LIN {X 0,Y 482.021,Z 1133.799,A -85,B 0,C 180,E1 13794.402,E2 13794.402} C_VEL
LIN {X 0,Y 488.852,Z 1107.216,A -85,B 0,C 180,E1 13800.271,E2 13800.271} C_VEL
LIN {X 0,Y 497.315,Z 1077.498,A -85,B 0,C 180,E1 13805.263,E2 13805.263} C_VEL
LIN {X 0,Y 507.512,Z 1042.761,A -85,B 0,C 180,E1 13809.804,E2 13809.804} C_VEL
LIN {X 0,Y 518.482,Z 1004.016,A -85,B 0,C 180,E1 13813.68,E2 13813.68} C_VEL
LIN {X 0,Y 529.347,Z 962.337,A -85,B 0,C 180,E1 13816.876,E2 13816.876} C_VEL
LIN {X 0,Y 539.035,Z 917.758,A -85,B 0,C 180,E1 13819.437,E2 13819.437} C_VEL
LIN {X 0,Y 545.481,Z 880.736,A -85,B 0,C 180,E1 13821.049,E2 13821.049} C_VEL
LIN {X 0,Y 530.255,Z 846.769,A -85,B 0,C 180,E1 13825.083,E2 13825.083} C_VEL
LIN {X 0,Y 514.025,Z 818.402,A -85,B 0,C 180,E1 13829.146,E2 13829.146} C_VEL
LIN {X 0,Y 498.472,Z 795.623,A -85,B 0,C 180,E1 13833.243,E2 13833.243} C_VEL
LIN {X 0,Y 488.833,Z 782.735,A -85,B 0,C 180,E1 13836.078,E2 13836.078} C_VEL
LIN {X 0,Y 483.89,Z 776.161,A -85,B 0,C 180,E1 13837.704,E2 13837.704} C_VEL
LIN {X 0,Y 479.927,Z 770.269,A -85,B 0,C 180,E1 13839.148,E2 13839.148} C_VEL
LIN {X 0,Y 474.71,Z 764.689,A -85,B 0,C 180,E1 13841.152,E2 13841.152} C_VEL
LIN {X 0,Y 474.293,Z 762.06,A -85,B 0,C 180,E1 13841.534,E2 13841.534} C_VEL
LIN {X 0,Y 474.67,Z 762.06,A -85,B 0,C 180,E1 13847.136,E2 13847.136} C_VEL
LIN {X 0,Y 475.044,Z 762.06,A -85,B 0,C 180,E1 13853.146,E2 13853.146} C_VEL
LIN {X 0,Y 475.398,Z 762.06,A -85,B 0,C 180,E1 13858.189,E2 13858.189} C_VEL
LIN {X 0,Y 475.263,Z 762.06,A -85,B 0,C 180,E1 13863.656,E2 13863.656} C_VEL
LIN {X 0,Y 474.96,Z 762.06,A -85,B 0,C 180,E1 13869.496,E2 13869.496} C_VEL
LIN {X 0,Y 474.723,Z 762.06,A -85,B 0,C 180,E1 13874.762,E2 13874.762} C_VEL
LIN {X 0,Y 474.615,Z 762.484,A -85,B 0,C 180,E1 13878.205,E2 13878.205} C_VEL
LIN {X 0,Y 476.602,Z 767.385,A -85,B 0,C 180,E1 13879.126,E2 13879.126} C_VEL
LIN {X 0,Y 480.342,Z 770.702,A -85,B 0,C 180,E1 13880.495,E2 13880.495} C_VEL
LIN {X 0,Y 484.534,Z 776.398,A -85,B 0,C 180,E1 13881.986,E2 13881.986} C_VEL
LIN {X 0,Y 496.6,Z 792.603,A -85,B 0,C 180,E1 13885.705,E2 13885.705} C_VEL
LIN {X 0,Y 513.454,Z 816.532,A -85,B 0,C 180,E1 13890.028,E2 13890.028} C_VEL
LIN {X 0,Y 531.553,Z 846.468,A -85,B 0,C 180,E1 13894.197,E2 13894.197} C_VEL
LIN {X 0,Y 547.68,Z 879.498,A -85,B 0,C 180,E1 13897.952,E2 13897.952} C_VEL
LIN {X 0,Y 548.07,Z 883.694,A -85,B 0,C 180,E1 13898.206,E2 13898.206} C_VEL
LIN {X 0,Y 540.632,Z 928.209,A -85,B 0,C 180,E1 13899.828,E2 13899.828} C_VEL
LIN {X 0,Y 531.328,Z 973.235,A -85,B 0,C 180,E1 13902.174,E2 13902.174} C_VEL
LIN {X 0,Y 520.612,Z 1017.117,A -85,B 0,C 180,E1 13905.219,E2 13905.219} C_VEL
LIN {X 0,Y 510.113,Z 1056.037,A -85,B 0,C 180,E1 13908.767,E2 13908.767} C_VEL
LIN {X 0,Y 499.446,Z 1094.323,A -85,B 0,C 180,E1 13913.266,E2 13913.266} C_VEL
LIN {X 0,Y 490.54,Z 1126.605,A -85,B 0,C 180,E1 13918.183,E2 13918.183} C_VEL
LIN {X 0,Y 483.623,Z 1154.685,A -85,B 0,C 180,E1 13923.669,E2 13923.669} C_VEL
LIN {X 0,Y 479.218,Z 1176.457,A -85,B 0,C 180,E1 13929.307,E2 13929.307} C_VEL
LIN {X 0,Y 476.873,Z 1192.347,A -85,B 0,C 180,E1 13934.876,E2 13934.876} C_VEL
LIN {X 0,Y 475.804,Z 1202.186,A -85,B 0,C 180,E1 13939.929,E2 13939.929} C_VEL
LIN {X 0,Y 475.654,Z 1204.167,A -85,B 0,C 180,E1 13941.356,E2 13941.356} C_VEL
LIN {X 0,Y 473.042,Z 1206.128,A -85,B 0,C 180,E1 13942.887,E2 13942.887} C_VEL
LIN {X 0,Y 467.509,Z 1208.379,A -85,B 0,C 180,E1 13945.396,E2 13945.396} C_VEL
LIN {X 0,Y 467.504,Z 1208.319,A -85,B 0,C 180,E1 13945.463,E2 13945.463} C_VEL
LIN {X 0,Y 467.695,Z 1210,A -85,B 0,C 180,E1 13949.999,E2 13949.999} C_VEL
LIN {X 0,Y 467.612,Z 1207.633,A -85,B 0,C 180,E1 13955.562,E2 13955.562} C_VEL
LIN {X 0,Y 468.046,Z 1200.643,A -85,B 0,C 180,E1 13961.169,E2 13961.169} C_VEL
LIN {X 0,Y 469.482,Z 1188.604,A -85,B 0,C 180,E1 13966.838,E2 13966.838} C_VEL
LIN {X 0,Y 472.232,Z 1172.652,A -85,B 0,C 180,E1 13972.122,E2 13972.122} C_VEL
LIN {X 0,Y 477.422,Z 1149.519,A -85,B 0,C 180,E1 13977.829,E2 13977.829} C_VEL
LIN {X 0,Y 484.963,Z 1121.457,A -85,B 0,C 180,E1 13983.186,E2 13983.186} C_VEL
LIN {X 0,Y 494.517,Z 1087.969,A -85,B 0,C 180,E1 13988.108,E2 13988.108} C_VEL
LIN {X 0,Y 505.375,Z 1050.696,A -85,B 0,C 180,E1 13992.39,E2 13992.39} C_VEL
LIN {X 0,Y 516.934,Z 1008.902,A -85,B 0,C 180,E1 13996.039,E2 13996.039} C_VEL
LIN {X 0,Y 527.27,Z 967.405,A -85,B 0,C 180,E1 13998.822,E2 13998.822} C_VEL
LIN {X 0,Y 536.686,Z 921.282,A -85,B 0,C 180,E1 14001.121,E2 14001.121} C_VEL
LIN {X 0,Y 542.571,Z 883.848,A -85,B 0,C 180,E1 14002.522,E2 14002.522} C_VEL
LIN {X 0,Y 527.23,Z 851.526,A -85,B 0,C 180,E1 14006.303,E2 14006.303} C_VEL
LIN {X 0,Y 509.607,Z 821.901,A -85,B 0,C 180,E1 14010.564,E2 14010.564} C_VEL
LIN {X 0,Y 492.359,Z 797.074,A -85,B 0,C 180,E1 14015.213,E2 14015.213} C_VEL
LIN {X 0,Y 481.779,Z 783.224,A -85,B 0,C 180,E1 14018.607,E2 14018.607} C_VEL
LIN {X 0,Y 476.584,Z 776.309,A -85,B 0,C 180,E1 14020.545,E2 14020.545} C_VEL
LIN {X 0,Y 472.76,Z 771.079,A -85,B 0,C 180,E1 14022.135,E2 14022.135} C_VEL
LIN {X 0,Y 471.499,Z 769.36,A -85,B 0,C 180,E1 14022.696,E2 14022.696} C_VEL
LIN {X 0,Y 467.212,Z 764.911,A -85,B 0,C 180,E1 14024.695,E2 14024.695} C_VEL
LIN {X 0,Y 466.74,Z 762.06,A -85,B 0,C 180,E1 14025.152,E2 14025.152} C_VEL
LIN {X 0,Y 467.07,Z 762.06,A -85,B 0,C 180,E1 14030.681,E2 14030.681} C_VEL
LIN {X 0,Y 467.355,Z 762.06,A -85,B 0,C 180,E1 14036.282,E2 14036.282} C_VEL
LIN {X 0,Y 467.491,Z 762.06,A -85,B 0,C 180,E1 14041.841,E2 14041.841} C_VEL
LIN {X 0,Y 467.171,Z 762.06,A -85,B 0,C 180,E1 14047.422,E2 14047.422} C_VEL
LIN {X 0,Y 466.641,Z 762.06,A -85,B 0,C 180,E1 14053.72,E2 14053.72} C_VEL
LIN {X 0,Y 466.542,Z 762.875,A -85,B 0,C 180,E1 14055.305,E2 14055.305} C_VEL
LIN {X 0,Y 468.796,Z 767.622,A -85,B 0,C 180,E1 14056.55,E2 14056.55} C_VEL
LIN {X 0,Y 472.464,Z 770.774,A -85,B 0,C 180,E1 14058.157,E2 14058.157} C_VEL
LIN {X 0,Y 476.384,Z 776.273,A -85,B 0,C 180,E1 14059.803,E2 14059.803} C_VEL
LIN {X 0,Y 478.642,Z 779.134,A -85,B 0,C 180,E1 14060.669,E2 14060.669} C_VEL
LIN {X 0,Y 484.508,Z 786.882,A -85,B 0,C 180,E1 14062.75,E2 14062.75} C_VEL
LIN {X 0,Y 494.565,Z 800.367,A -85,B 0,C 180,E1 14065.895,E2 14065.895} C_VEL
LIN {X 0,Y 509.773,Z 823.065,A -85,B 0,C 180,E1 14070.123,E2 14070.123} C_VEL
LIN {X 0,Y 525.508,Z 851.418,A -85,B 0,C 180,E1 14074.276,E2 14074.276} C_VEL
LIN {X 0,Y 539.633,Z 883.823,A -85,B 0,C 180,E1 14078.242,E2 14078.242} C_VEL
LIN {X 0,Y 539.67,Z 888.681,A -85,B 0,C 180,E1 14078.535,E2 14078.535} C_VEL
LIN {X 0,Y 531.251,Z 930.768,A -85,B 0,C 180,E1 14080.477,E2 14080.477} C_VEL
LIN {X 0,Y 520.428,Z 975.76,A -85,B 0,C 180,E1 14083.297,E2 14083.297} C_VEL
LIN {X 0,Y 509.34,Z 1015.639,A -85,B 0,C 180,E1 14086.633,E2 14086.633} C_VEL
LIN {X 0,Y 497.817,Z 1054.175,A -85,B 0,C 180,E1 14090.841,E2 14090.841} C_VEL
LIN {X 0,Y 487.835,Z 1086.765,A -85,B 0,C 180,E1 14095.486,E2 14095.486} C_VEL
LIN {X 0,Y 479.242,Z 1116.664,A -85,B 0,C 180,E1 14101.002,E2 14101.002} C_VEL
LIN {X 0,Y 473.034,Z 1140.832,A -85,B 0,C 180,E1 14106.964,E2 14106.964} C_VEL
LIN {X 0,Y 469.704,Z 1158.095,A -85,B 0,C 180,E1 14112.688,E2 14112.688} C_VEL
LIN {X 0,Y 468.161,Z 1169.156,A -85,B 0,C 180,E1 14117.89,E2 14117.89} C_VEL
LIN {X 0,Y 467.701,Z 1175.956,A -85,B 0,C 180,E1 14122.575,E2 14122.575} C_VEL
LIN {X 0,Y 467.42,Z 1179.674,A -85,B 0,C 180,E1 14128.148,E2 14128.148} C_VEL
LIN {X 0,Y 467.598,Z 1179.656,A -85,B 0,C 180,E1 14131.853,E2 14131.853} C_VEL
LIN {X 0,Y 467.744,Z 1175.86,A -85,B 0,C 180,E1 14137.426,E2 14137.426} C_VEL
LIN {X 0,Y 468.381,Z 1167.229,A -85,B 0,C 180,E1 14143.053,E2 14143.053} C_VEL
LIN {X 0,Y 470.371,Z 1153.967,A -85,B 0,C 180,E1 14148.74,E2 14148.74} C_VEL
LIN {X 0,Y 474.261,Z 1135.424,A -85,B 0,C 180,E1 14154.471,E2 14154.471} C_VEL
LIN {X 0,Y 480.847,Z 1110.384,A -85,B 0,C 180,E1 14160.188,E2 14160.188} C_VEL
LIN {X 0,Y 489.563,Z 1081.41,A -85,B 0,C 180,E1 14165.278,E2 14165.278} C_VEL
LIN {X 0,Y 500.064,Z 1046.801,A -85,B 0,C 180,E1 14169.953,E2 14169.953} C_VEL
LIN {X 0,Y 511,Z 1010.288,A -85,B 0,C 180,E1 14173.776,E2 14173.776} C_VEL
LIN {X 0,Y 522.097,Z 969.271,A -85,B 0,C 180,E1 14177.06,E2 14177.06} C_VEL
LIN {X 0,Y 532.581,Z 924.406,A -85,B 0,C 180,E1 14179.779,E2 14179.779} C_VEL
LIN {X 0,Y 539.912,Z 884.236,A -85,B 0,C 180,E1 14181.599,E2 14181.599} C_VEL
LIN {X 0,Y 525.577,Z 851.517,A -85,B 0,C 180,E1 14185.604,E2 14185.604} C_VEL
LIN {X 0,Y 509.447,Z 822.562,A -85,B 0,C 180,E1 14189.851,E2 14189.851} C_VEL
LIN {X 0,Y 492.461,Z 797.228,A -85,B 0,C 180,E1 14194.62,E2 14194.62} C_VEL
LIN {X 0,Y 481.516,Z 783.139,A -85,B 0,C 180,E1 14198.134,E2 14198.134} C_VEL
LIN {X 0,Y 476.61,Z 776.434,A -85,B 0,C 180,E1 14199.965,E2 14199.965} C_VEL
LIN {X 0,Y 472.601,Z 771.322,A -85,B 0,C 180,E1 14201.608,E2 14201.608} C_VEL
LIN {X 0,Y 471.105,Z 769.289,A -85,B 0,C 180,E1 14202.272,E2 14202.272} C_VEL
LIN {X 0,Y 466.951,Z 764.704,A -85,B 0,C 180,E1 14204.228,E2 14204.228} C_VEL
LIN {X 0,Y 466.521,Z 762.06,A -85,B 0,C 180,E1 14204.754,E2 14204.754} C_VEL
LIN {X 0,Y 467.085,Z 762.06,A -85,B 0,C 180,E1 14210.703,E2 14210.703} C_VEL
LIN {X 0,Y 467.468,Z 762.06,A -85,B 0,C 180,E1 14216.304,E2 14216.304} C_VEL
LIN {X 0,Y 467.528,Z 762.06,A -85,B 0,C 180,E1 14221.863,E2 14221.863} C_VEL
LIN {X 0,Y 467.151,Z 762.06,A -85,B 0,C 180,E1 14227.444,E2 14227.444} C_VEL
LIN {X 0,Y 466.808,Z 762.06,A -85,B 0,C 180,E1 14233.796,E2 14233.796} C_VEL
LIN {X 0,Y 466.809,Z 762.508,A -85,B 0,C 180,E1 14235.078,E2 14235.078} C_VEL
LIN {X 0,Y 468.581,Z 767.145,A -85,B 0,C 180,E1 14236.098,E2 14236.098} C_VEL
LIN {X 0,Y 472.763,Z 770.814,A -85,B 0,C 180,E1 14237.921,E2 14237.921} C_VEL
LIN {X 0,Y 476.444,Z 776.177,A -85,B 0,C 180,E1 14239.461,E2 14239.461} C_VEL
LIN {X 0,Y 478.596,Z 778.637,A -85,B 0,C 180,E1 14240.271,E2 14240.271} C_VEL
LIN {X 0,Y 484.917,Z 787.333,A -85,B 0,C 180,E1 14242.51,E2 14242.51} C_VEL
LIN {X 0,Y 494.366,Z 799.789,A -85,B 0,C 180,E1 14245.405,E2 14245.405} C_VEL
LIN {X 0,Y 510.644,Z 823.428,A -85,B 0,C 180,E1 14249.711,E2 14249.711} C_VEL
LIN {X 0,Y 527.987,Z 853.064,A -85,B 0,C 180,E1 14253.901,E2 14253.901} C_VEL
LIN {X 0,Y 542.933,Z 884.677,A -85,B 0,C 180,E1 14257.574,E2 14257.574} C_VEL
LIN {X 0,Y 535.142,Z 929.856,A -85,B 0,C 180,E1 14259.248,E2 14259.248} C_VEL
LIN {X 0,Y 525.063,Z 976.261,A -85,B 0,C 180,E1 14261.713,E2 14261.713} C_VEL
LIN {X 0,Y 514.211,Z 1019.181,A -85,B 0,C 180,E1 14264.76,E2 14264.76} C_VEL
LIN {X 0,Y 502.972,Z 1058.986,A -85,B 0,C 180,E1 14268.487,E2 14268.487} C_VEL
LIN {X 0,Y 492.202,Z 1096.115,A -85,B 0,C 180,E1 14272.969,E2 14272.969} C_VEL
LIN {X 0,Y 482.385,Z 1130.255,A -85,B 0,C 180,E1 14278.35,E2 14278.35} C_VEL
LIN {X 0,Y 475.817,Z 1155.975,A -85,B 0,C 180,E1 14283.6,E2 14283.6} C_VEL
LIN {X 0,Y 471.294,Z 1177.475,A -85,B 0,C 180,E1 14289.347,E2 14289.347} C_VEL
LIN {X 0,Y 468.888,Z 1193.647,A -85,B 0,C 180,E1 14295.215,E2 14295.215} C_VEL
LIN {X 0,Y 467.832,Z 1203.513,A -85,B 0,C 180,E1 14300.705,E2 14300.705} C_VEL
LIN {X 0,Y 467.504,Z 1208.319,A -85,B 0,C 180,E1 14305.463,E2 14305.463} C_VEL
LIN {X 0,Y 464.981,Z 1209.328,A -85,B 0,C 180,E1 14307.044,E2 14307.044} C_VEL
LIN {X 0,Y 459.785,Z 1209.902,A -85,B 0,C 180,E1 14309.422,E2 14309.422} C_VEL
LIN {X 0,Y 459.736,Z 1209.946,A -85,B 0,C 180,E1 14309.696,E2 14309.696} C_VEL
LIN {X 0,Y 459.672,Z 1208.874,A -85,B 0,C 180,E1 14313.769,E2 14313.769} C_VEL
LIN {X 0,Y 459.913,Z 1204.668,A -85,B 0,C 180,E1 14318.502,E2 14318.502} C_VEL
LIN {X 0,Y 460.737,Z 1195.374,A -85,B 0,C 180,E1 14324.073,E2 14324.073} C_VEL
LIN {X 0,Y 463.106,Z 1180.326,A -85,B 0,C 180,E1 14330.035,E2 14330.035} C_VEL
LIN {X 0,Y 467.49,Z 1159.685,A -85,B 0,C 180,E1 14335.871,E2 14335.871} C_VEL
LIN {X 0,Y 474.645,Z 1132.681,A -85,B 0,C 180,E1 14341.688,E2 14341.688} C_VEL
LIN {X 0,Y 484.107,Z 1100.414,A -85,B 0,C 180,E1 14346.965,E2 14346.965} C_VEL
LIN {X 0,Y 494.946,Z 1064.966,A -85,B 0,C 180,E1 14351.478,E2 14351.478} C_VEL
LIN {X 0,Y 507.001,Z 1023.879,A -85,B 0,C 180,E1 14355.476,E2 14355.476} C_VEL
LIN {X 0,Y 517.974,Z 982.943,A -85,B 0,C 180,E1 14358.536,E2 14358.536} C_VEL
LIN {X 0,Y 529.125,Z 934.201,A -85,B 0,C 180,E1 14361.211,E2 14361.211} C_VEL
LIN {X 0,Y 537.157,Z 887.442,A -85,B 0,C 180,E1 14363.086,E2 14363.086} C_VEL
LIN {X 0,Y 522.309,Z 855.549,A -85,B 0,C 180,E1 14366.916,E2 14366.916} C_VEL
LIN {X 0,Y 505.838,Z 827.369,A -85,B 0,C 180,E1 14371.135,E2 14371.135} C_VEL
LIN {X 0,Y 489.999,Z 804.007,A -85,B 0,C 180,E1 14375.571,E2 14375.571} C_VEL
LIN {X 0,Y 479.443,Z 790.095,A -85,B 0,C 180,E1 14379.043,E2 14379.043} C_VEL
LIN {X 0,Y 474.776,Z 783.74,A -85,B 0,C 180,E1 14380.83,E2 14380.83} C_VEL
LIN {X 0,Y 470.687,Z 777.697,A -85,B 0,C 180,E1 14382.595,E2 14382.595} C_VEL
LIN {X 0,Y 465.499,Z 772.049,A -85,B 0,C 180,E1 14385.056,E2 14385.056} C_VEL
LIN {X 0,Y 464.758,Z 769.685,A -85,B 0,C 180,E1 14385.538,E2 14385.538} C_VEL
LIN {X 0,Y 459.786,Z 765.515,A -85,B 0,C 180,E1 14388.437,E2 14388.437} C_VEL
LIN {X 0,Y 459.057,Z 762.06,A -85,B 0,C 180,E1 14389.32,E2 14389.32} C_VEL
LIN {X 0,Y 459.365,Z 762.06,A -85,B 0,C 180,E1 14394.326,E2 14394.326} C_VEL
LIN {X 0,Y 459.759,Z 762.06,A -85,B 0,C 180,E1 14399.989,E2 14399.989} C_VEL
LIN {X 0,Y 459.408,Z 762.06,A -85,B 0,C 180,E1 14405.651,E2 14405.651} C_VEL
LIN {X 0,Y 459.012,Z 762.388,A -85,B 0,C 180,E1 14411.259,E2 14411.259} C_VEL
LIN {X 0,Y 460.474,Z 766.901,A -85,B 0,C 180,E1 14412.484,E2 14412.484} C_VEL
LIN {X 0,Y 464.855,Z 770.601,A -85,B 0,C 180,E1 14414.98,E2 14414.98} C_VEL
LIN {X 0,Y 468.212,Z 775.992,A -85,B 0,C 180,E1 14416.752,E2 14416.752} C_VEL
LIN {X 0,Y 470.825,Z 778.622,A -85,B 0,C 180,E1 14417.92,E2 14417.92} C_VEL
LIN {X 0,Y 475.459,Z 784.284,A -85,B 0,C 180,E1 14419.843,E2 14419.843} C_VEL
LIN {X 0,Y 488.256,Z 802.049,A -85,B 0,C 180,E1 14424.377,E2 14424.377} C_VEL
LIN {X 0,Y 501.005,Z 820.808,A -85,B 0,C 180,E1 14428.215,E2 14428.215} C_VEL
LIN {X 0,Y 516.276,Z 847.033,A -85,B 0,C 180,E1 14432.492,E2 14432.492} C_VEL
LIN {X 0,Y 530.399,Z 877.971,A -85,B 0,C 180,E1 14436.566,E2 14436.566} C_VEL
LIN {X 0,Y 534.534,Z 889.963,A -85,B 0,C 180,E1 14437.908,E2 14437.908} C_VEL
LIN {X 0,Y 525.762,Z 932.379,A -85,B 0,C 180,E1 14439.886,E2 14439.886} C_VEL
LIN {X 0,Y 514.844,Z 976.225,A -85,B 0,C 180,E1 14442.655,E2 14442.655} C_VEL
LIN {X 0,Y 503.09,Z 1017.032,A -85,B 0,C 180,E1 14446.105,E2 14446.105} C_VEL
LIN {X 0,Y 491.121,Z 1055.632,A -85,B 0,C 180,E1 14450.383,E2 14450.383} C_VEL
LIN {X 0,Y 480.429,Z 1089.06,A -85,B 0,C 180,E1 14455.266,E2 14455.266} C_VEL
LIN {X 0,Y 472.214,Z 1116.276,A -85,B 0,C 180,E1 14460.379,E2 14460.379} C_VEL
LIN {X 0,Y 465.927,Z 1139.404,A -85,B 0,C 180,E1 14466.085,E2 14466.085} C_VEL
LIN {X 0,Y 462.151,Z 1157.539,A -85,B 0,C 180,E1 14472.077,E2 14472.077} C_VEL
LIN {X 0,Y 460.321,Z 1169.407,A -85,B 0,C 180,E1 14477.681,E2 14477.681} C_VEL
LIN {X 0,Y 459.807,Z 1176.007,A -85,B 0,C 180,E1 14482.447,E2 14482.447} C_VEL
LIN {X 0,Y 459.517,Z 1179.673,A -85,B 0,C 180,E1 14488.116,E2 14488.116} C_VEL
LIN {X 0,Y 459.691,Z 1179.656,A -85,B 0,C 180,E1 14491.885,E2 14491.885} C_VEL
LIN {X 0,Y 459.852,Z 1175.916,A -85,B 0,C 180,E1 14497.554,E2 14497.554} C_VEL
LIN {X 0,Y 460.564,Z 1167.494,A -85,B 0,C 180,E1 14503.279,E2 14503.279} C_VEL
LIN {X 0,Y 462.682,Z 1154.236,A -85,B 0,C 180,E1 14509.063,E2 14509.063} C_VEL
LIN {X 0,Y 466.844,Z 1135.695,A -85,B 0,C 180,E1 14514.886,E2 14514.886} C_VEL
LIN {X 0,Y 474.217,Z 1109.478,A -85,B 0,C 180,E1 14520.92,E2 14520.92} C_VEL
LIN {X 0,Y 483.373,Z 1079.927,A -85,B 0,C 180,E1 14526.108,E2 14526.108} C_VEL
LIN {X 0,Y 494.425,Z 1045.238,A -85,B 0,C 180,E1 14530.783,E2 14530.783} C_VEL
LIN {X 0,Y 505.798,Z 1008.274,A -85,B 0,C 180,E1 14534.619,E2 14534.619} C_VEL
LIN {X 0,Y 517.301,Z 967.146,A -85,B 0,C 180,E1 14537.88,E2 14537.88} C_VEL
LIN {X 0,Y 527.574,Z 924.051,A -85,B 0,C 180,E1 14540.474,E2 14540.474} C_VEL
LIN {X 0,Y 534.465,Z 887.885,A -85,B 0,C 180,E1 14542.141,E2 14542.141} C_VEL
LIN {X 0,Y 520.643,Z 855.794,A -85,B 0,C 180,E1 14546.175,E2 14546.175} C_VEL
LIN {X 0,Y 505.438,Z 827.967,A -85,B 0,C 180,E1 14550.414,E2 14550.414} C_VEL
LIN {X 0,Y 489.726,Z 803.978,A -85,B 0,C 180,E1 14555.035,E2 14555.035} C_VEL
LIN {X 0,Y 479.336,Z 790.149,A -85,B 0,C 180,E1 14558.515,E2 14558.515} C_VEL
LIN {X 0,Y 474.508,Z 783.671,A -85,B 0,C 180,E1 14560.358,E2 14560.358} C_VEL
LIN {X 0,Y 470.417,Z 777.61,A -85,B 0,C 180,E1 14562.125,E2 14562.125} C_VEL
LIN {X 0,Y 465.226,Z 771.897,A -85,B 0,C 180,E1 14564.59,E2 14564.59} C_VEL
LIN {X 0,Y 464.131,Z 769.564,A -85,B 0,C 180,E1 14565.239,E2 14565.239} C_VEL
LIN {X 0,Y 459.461,Z 765.025,A -85,B 0,C 180,E1 14568.03,E2 14568.03} C_VEL
LIN {X 0,Y 458.988,Z 762.06,A -85,B 0,C 180,E1 14568.62,E2 14568.62} C_VEL
LIN {X 0,Y 459.36,Z 762.06,A -85,B 0,C 180,E1 14574.348,E2 14574.348} C_VEL
LIN {X 0,Y 459.775,Z 762.06,A -85,B 0,C 180,E1 14580.011,E2 14580.011} C_VEL
LIN {X 0,Y 459.366,Z 762.06,A -85,B 0,C 180,E1 14585.674,E2 14585.674} C_VEL
LIN {X 0,Y 459.087,Z 762.498,A -85,B 0,C 180,E1 14591.04,E2 14591.04} C_VEL
LIN {X 0,Y 460.872,Z 767.231,A -85,B 0,C 180,E1 14592.435,E2 14592.435} C_VEL
LIN {X 0,Y 465.092,Z 770.623,A -85,B 0,C 180,E1 14594.768,E2 14594.768} C_VEL
LIN {X 0,Y 468.478,Z 776.017,A -85,B 0,C 180,E1 14596.523,E2 14596.523} C_VEL
LIN {X 0,Y 471.01,Z 778.412,A -85,B 0,C 180,E1 14597.633,E2 14597.633} C_VEL
LIN {X 0,Y 475.518,Z 784.176,A -85,B 0,C 180,E1 14599.5,E2 14599.5} C_VEL
LIN {X 0,Y 487.699,Z 800.88,A -85,B 0,C 180,E1 14603.761,E2 14603.761} C_VEL
LIN {X 0,Y 502.204,Z 821.682,A -85,B 0,C 180,E1 14607.938,E2 14607.938} C_VEL
LIN {X 0,Y 519.434,Z 850.037,A -85,B 0,C 180,E1 14612.35,E2 14612.35} C_VEL
LIN {X 0,Y 535.88,Z 884.202,A -85,B 0,C 180,E1 14616.579,E2 14616.579} C_VEL
LIN {X 0,Y 537.377,Z 889.447,A -85,B 0,C 180,E1 14617.054,E2 14617.054} C_VEL
LIN {X 0,Y 529.104,Z 934.2,A -85,B 0,C 180,E1 14618.792,E2 14618.792} C_VEL
LIN {X 0,Y 518.434,Z 981.141,A -85,B 0,C 180,E1 14621.361,E2 14621.361} C_VEL
LIN {X 0,Y 507.485,Z 1022.217,A -85,B 0,C 180,E1 14624.386,E2 14624.386} C_VEL
LIN {X 0,Y 495.904,Z 1061.61,A -85,B 0,C 180,E1 14628.161,E2 14628.161} C_VEL
LIN {X 0,Y 485.242,Z 1096.941,A -85,B 0,C 180,E1 14632.537,E2 14632.537} C_VEL
LIN {X 0,Y 475.31,Z 1129.981,A -85,B 0,C 180,E1 14637.823,E2 14637.823} C_VEL
LIN {X 0,Y 468.393,Z 1155.702,A -85,B 0,C 180,E1 14643.149,E2 14643.149} C_VEL
LIN {X 0,Y 463.612,Z 1177.205,A -85,B 0,C 180,E1 14648.989,E2 14648.989} C_VEL
LIN {X 0,Y 461.095,Z 1193.034,A -85,B 0,C 180,E1 14654.8,E2 14654.8} C_VEL
LIN {X 0,Y 459.94,Z 1203.419,A -85,B 0,C 180,E1 14660.544,E2 14660.544} C_VEL
LIN {X 0,Y 459.599,Z 1208.369,A -85,B 0,C 180,E1 14665.465,E2 14665.465} C_VEL
LIN {X 0,Y 459.736,Z 1209.946,A -85,B 0,C 180,E1 14669.696,E2 14669.696} C_VEL
LIN {X 0,Y 457.353,Z 1209.886,A -85,B 0,C 180,E1 14671.305,E2 14671.305} C_VEL
LIN {X 0,Y 451.771,Z 1208.578,A -85,B 0,C 180,E1 14673.995,E2 14673.995} C_VEL
LIN {X 0,Y 452.069,Z 1203.161,A -85,B 0,C 180,E1 14679.62,E2 14679.62} C_VEL
LIN {X 0,Y 453.258,Z 1192.772,A -85,B 0,C 180,E1 14685.468,E2 14685.468} C_VEL
LIN {X 0,Y 455.955,Z 1176.943,A -85,B 0,C 180,E1 14691.379,E2 14691.379} C_VEL
LIN {X 0,Y 460.984,Z 1155.429,A -85,B 0,C 180,E1 14697.316,E2 14697.316} C_VEL
LIN {X 0,Y 468.753,Z 1128.396,A -85,B 0,C 180,E1 14702.95,E2 14702.95} C_VEL
LIN {X 0,Y 479.163,Z 1095.224,A -85,B 0,C 180,E1 14708.279,E2 14708.279} C_VEL
LIN {X 0,Y 490.331,Z 1059.502,A -85,B 0,C 180,E1 14712.686,E2 14712.686} C_VEL
LIN {X 0,Y 502.865,Z 1018.462,A -85,B 0,C 180,E1 14716.586,E2 14716.586} C_VEL
LIN {X 0,Y 514.507,Z 975.337,A -85,B 0,C 180,E1 14719.666,E2 14719.666} C_VEL
LIN {X 0,Y 525.319,Z 928.259,A -85,B 0,C 180,E1 14722.167,E2 14722.167} C_VEL
LIN {X 0,Y 532.13,Z 891.783,A -85,B 0,C 180,E1 14723.562,E2 14723.562} C_VEL
LIN {X 0,Y 517.239,Z 859.358,A -85,B 0,C 180,E1 14727.587,E2 14727.587} C_VEL
LIN {X 0,Y 501.801,Z 832.39,A -85,B 0,C 180,E1 14731.756,E2 14731.756} C_VEL
LIN {X 0,Y 487.096,Z 810.37,A -85,B 0,C 180,E1 14736.082,E2 14736.082} C_VEL
LIN {X 0,Y 477.134,Z 796.971,A -85,B 0,C 180,E1 14739.482,E2 14739.482} C_VEL
LIN {X 0,Y 472.566,Z 790.771,A -85,B 0,C 180,E1 14741.282,E2 14741.282} C_VEL
LIN {X 0,Y 467.697,Z 784.149,A -85,B 0,C 180,E1 14743.448,E2 14743.448} C_VEL
LIN {X 0,Y 463.522,Z 778.425,A -85,B 0,C 180,E1 14745.597,E2 14745.597} C_VEL
LIN {X 0,Y 458.058,Z 772.051,A -85,B 0,C 180,E1 14748.995,E2 14748.995} C_VEL
LIN {X 0,Y 457.521,Z 769.809,A -85,B 0,C 180,E1 14749.524,E2 14749.524} C_VEL
LIN {X 0,Y 451.937,Z 764.768,A -85,B 0,C 180,E1 14755.194,E2 14755.194} C_VEL
LIN {X 0,Y 451.543,Z 762.06,A -85,B 0,C 180,E1 14756.632,E2 14756.632} C_VEL
LIN {X 0,Y 451.699,Z 762.06,A -85,B 0,C 180,E1 14761.906,E2 14761.906} C_VEL
LIN {X 0,Y 451.618,Z 762.689,A -85,B 0,C 180,E1 14764.306,E2 14764.306} C_VEL
LIN {X 0,Y 454.334,Z 768.286,A -85,B 0,C 180,E1 14768.331,E2 14768.331} C_VEL
LIN {X 0,Y 457.573,Z 770.624,A -85,B 0,C 180,E1 14770.994,E2 14770.994} C_VEL
LIN {X 0,Y 460.337,Z 775.756,A -85,B 0,C 180,E1 14773.03,E2 14773.03} C_VEL
LIN {X 0,Y 463.367,Z 778.452,A -85,B 0,C 180,E1 14774.747,E2 14774.747} C_VEL
LIN {X 0,Y 467.52,Z 784.178,A -85,B 0,C 180,E1 14776.898,E2 14776.898} C_VEL
LIN {X 0,Y 470.033,Z 787.867,A -85,B 0,C 180,E1 14778.072,E2 14778.072} C_VEL
LIN {X 0,Y 475.252,Z 794.403,A -85,B 0,C 180,E1 14780.216,E2 14780.216} C_VEL
LIN {X 0,Y 484.874,Z 807.458,A -85,B 0,C 180,E1 14783.704,E2 14783.704} C_VEL
LIN {X 0,Y 499.036,Z 829.015,A -85,B 0,C 180,E1 14788.176,E2 14788.176} C_VEL
LIN {X 0,Y 514.041,Z 856.405,A -85,B 0,C 180,E1 14792.616,E2 14792.616} C_VEL
LIN {X 0,Y 527.344,Z 887.392,A -85,B 0,C 180,E1 14796.697,E2 14796.697} C_VEL
LIN {X 0,Y 529.028,Z 893.334,A -85,B 0,C 180,E1 14797.354,E2 14797.354} C_VEL
LIN {X 0,Y 519.844,Z 936.207,A -85,B 0,C 180,E1 14799.411,E2 14799.411} C_VEL
LIN {X 0,Y 508.661,Z 979.359,A -85,B 0,C 180,E1 14802.199,E2 14802.199} C_VEL
LIN {X 0,Y 496.002,Z 1021.296,A -85,B 0,C 180,E1 14805.85,E2 14805.85} C_VEL
LIN {X 0,Y 484.409,Z 1057.183,A -85,B 0,C 180,E1 14809.935,E2 14809.935} C_VEL
LIN {X 0,Y 473.255,Z 1090.647,A -85,B 0,C 180,E1 14814.919,E2 14814.919} C_VEL
LIN {X 0,Y 464.451,Z 1118.672,A -85,B 0,C 180,E1 14820.358,E2 14820.358} C_VEL
LIN {X 0,Y 457.604,Z 1143.059,A -85,B 0,C 180,E1 14826.656,E2 14826.656} C_VEL
LIN {X 0,Y 454.028,Z 1159.737,A -85,B 0,C 180,E1 14832.571,E2 14832.571} C_VEL
LIN {X 0,Y 452.299,Z 1171.183,A -85,B 0,C 180,E1 14838.437,E2 14838.437} C_VEL
LIN {X 0,Y 451.735,Z 1177.933,A -85,B 0,C 180,E1 14844.241,E2 14844.241} C_VEL
LIN {X 0,Y 451.786,Z 1180.185,A -85,B 0,C 180,E1 14850.001,E2 14850.001} C_VEL
LIN {X 0,Y 451.79,Z 1177.85,A -85,B 0,C 180,E1 14855.76,E2 14855.76} C_VEL
LIN {X 0,Y 452.345,Z 1171.039,A -85,B 0,C 180,E1 14861.563,E2 14861.563} C_VEL
LIN {X 0,Y 454.107,Z 1159.528,A -85,B 0,C 180,E1 14867.428,E2 14867.428} C_VEL
LIN {X 0,Y 457.688,Z 1142.757,A -85,B 0,C 180,E1 14873.341,E2 14873.341} C_VEL
LIN {X 0,Y 464.471,Z 1118.251,A -85,B 0,C 180,E1 14879.659,E2 14879.659} C_VEL
LIN {X 0,Y 473.436,Z 1090.165,A -85,B 0,C 180,E1 14885.067,E2 14885.067} C_VEL
LIN {X 0,Y 484.835,Z 1056.067,A -85,B 0,C 180,E1 14890.115,E2 14890.115} C_VEL
LIN {X 0,Y 497.048,Z 1018.082,A -85,B 0,C 180,E1 14894.367,E2 14894.367} C_VEL
LIN {X 0,Y 508.943,Z 978.42,A -85,B 0,C 180,E1 14897.771,E2 14897.771} C_VEL
LIN {X 0,Y 520.354,Z 933.446,A -85,B 0,C 180,E1 14900.664,E2 14900.664} C_VEL
LIN {X 0,Y 529.063,Z 891.817,A -85,B 0,C 180,E1 14902.649,E2 14902.649} C_VEL
LIN {X 0,Y 515.431,Z 859.33,A -85,B 0,C 180,E1 14906.858,E2 14906.858} C_VEL
LIN {X 0,Y 500.559,Z 831.68,A -85,B 0,C 180,E1 14911.256,E2 14911.256} C_VEL
LIN {X 0,Y 486.455,Z 809.923,A -85,B 0,C 180,E1 14915.636,E2 14915.636} C_VEL
LIN {X 0,Y 477.024,Z 797.056,A -85,B 0,C 180,E1 14918.941,E2 14918.941} C_VEL
LIN {X 0,Y 472.438,Z 790.828,A -85,B 0,C 180,E1 14920.754,E2 14920.754} C_VEL
LIN {X 0,Y 467.422,Z 784.115,A -85,B 0,C 180,E1 14922.977,E2 14922.977} C_VEL
LIN {X 0,Y 463.348,Z 778.514,A -85,B 0,C 180,E1 14925.071,E2 14925.071} C_VEL
LIN {X 0,Y 457.809,Z 771.742,A -85,B 0,C 180,E1 14928.53,E2 14928.53} C_VEL
LIN {X 0,Y 457.239,Z 769.765,A -85,B 0,C 180,E1 14929.058,E2 14929.058} C_VEL
LIN {X 0,Y 451.946,Z 764.794,A -85,B 0,C 180,E1 14934.315,E2 14934.315} C_VEL
LIN {X 0,Y 451.546,Z 762.06,A -85,B 0,C 180,E1 14935.693,E2 14935.693} C_VEL
LIN {X 0,Y 451.725,Z 762.06,A -85,B 0,C 180,E1 14941.928,E2 14941.928} C_VEL
LIN {X 0,Y 451.532,Z 762.79,A -85,B 0,C 180,E1 14944.209,E2 14944.209} C_VEL
LIN {X 0,Y 454.746,Z 768.615,A -85,B 0,C 180,E1 14948.501,E2 14948.501} C_VEL
LIN {X 0,Y 457.722,Z 770.78,A -85,B 0,C 180,E1 14950.832,E2 14950.832} C_VEL
LIN {X 0,Y 460.675,Z 775.934,A -85,B 0,C 180,E1 14952.922,E2 14952.922} C_VEL
LIN {X 0,Y 463.569,Z 778.441,A -85,B 0,C 180,E1 14954.522,E2 14954.522} C_VEL
LIN {X 0,Y 467.791,Z 784.176,A -85,B 0,C 180,E1 14956.669,E2 14956.669} C_VEL
LIN {X 0,Y 470.332,Z 787.951,A -85,B 0,C 180,E1 14957.841,E2 14957.841} C_VEL
LIN {X 0,Y 475.32,Z 794.243,A -85,B 0,C 180,E1 14959.872,E2 14959.872} C_VEL
LIN {X 0,Y 485.543,Z 808.042,A -85,B 0,C 180,E1 14963.448,E2 14963.448} C_VEL
LIN {X 0,Y 500.855,Z 830.453,A -85,B 0,C 180,E1 14967.981,E2 14967.981} C_VEL
LIN {X 0,Y 517.186,Z 859.304,A -85,B 0,C 180,E1 14972.417,E2 14972.417} C_VEL
LIN {X 0,Y 532.101,Z 891.662,A -85,B 0,C 180,E1 14976.435,E2 14976.435} C_VEL
LIN {X 0,Y 522.978,Z 939.007,A -85,B 0,C 180,E1 14978.345,E2 14978.345} C_VEL
LIN {X 0,Y 512.26,Z 984.248,A -85,B 0,C 180,E1 14980.894,E2 14980.894} C_VEL
LIN {X 0,Y 500.414,Z 1026.622,A -85,B 0,C 180,E1 14984.124,E2 14984.124} C_VEL
LIN {X 0,Y 488.688,Z 1065.032,A -85,B 0,C 180,E1 14987.92,E2 14987.92} C_VEL
LIN {X 0,Y 477.159,Z 1101.161,A -85,B 0,C 180,E1 14992.585,E2 14992.585} C_VEL
LIN {X 0,Y 467.404,Z 1132.729,A -85,B 0,C 180,E1 14997.832,E2 14997.832} C_VEL
LIN {X 0,Y 459.99,Z 1159.407,A -85,B 0,C 180,E1 15003.672,E2 15003.672} C_VEL
LIN {X 0,Y 455.375,Z 1180.047,A -85,B 0,C 180,E1 15009.608,E2 15009.608} C_VEL
LIN {X 0,Y 452.873,Z 1195.566,A -85,B 0,C 180,E1 15015.905,E2 15015.905} C_VEL
LIN {X 0,Y 452.03,Z 1204.402,A -85,B 0,C 180,E1 15021.347,E2 15021.347} C_VEL
LIN {X 0,Y 451.775,Z 1208.683,A -85,B 0,C 180,E1 15026.163,E2 15026.163} C_VEL
LIN {X 0,Y 451.904,Z 1209.849,A -85,B 0,C 180,E1 15029.999,E2 15029.999} C_VEL
LIN {X 0,Y 451.771,Z 1208.578,A -85,B 0,C 180,E1 15033.995,E2 15033.995} C_VEL
LIN {X 0,Y 447.847,Z 1206.978,A -85,B 0,C 180,E1 15036.153,E2 15036.153} C_VEL
LIN {X 0,Y 444.052,Z 1204.723,A -85,B 0,C 180,E1 15038.337,E2 15038.337} C_VEL
LIN {X 0,Y 445.037,Z 1195.305,A -85,B 0,C 180,E1 15044.346,E2 15044.346} C_VEL
LIN {X 0,Y 447.419,Z 1181.158,A -85,B 0,C 180,E1 15050.253,E2 15050.253} C_VEL
LIN {X 0,Y 452.107,Z 1161.124,A -85,B 0,C 180,E1 15056.286,E2 15056.286} C_VEL
LIN {X 0,Y 459.978,Z 1133.837,A -85,B 0,C 180,E1 15062.437,E2 15062.437} C_VEL
LIN {X 0,Y 469.772,Z 1103.312,A -85,B 0,C 180,E1 15067.673,E2 15067.673} C_VEL
LIN {X 0,Y 482.013,Z 1066.392,A -85,B 0,C 180,E1 15072.559,E2 15072.559} C_VEL
LIN {X 0,Y 494.043,Z 1028.406,A -85,B 0,C 180,E1 15076.392,E2 15076.392} C_VEL
LIN {X 0,Y 506.496,Z 985.467,A -85,B 0,C 180,E1 15079.713,E2 15079.713} C_VEL
LIN {X 0,Y 517.77,Z 939.926,A -85,B 0,C 180,E1 15082.303,E2 15082.303} C_VEL
LIN {X 0,Y 526.466,Z 894.645,A -85,B 0,C 180,E1 15084.209,E2 15084.209} C_VEL
LIN {X 0,Y 511.773,Z 862.118,A -85,B 0,C 180,E1 15088.407,E2 15088.407} C_VEL
LIN {X 0,Y 496.475,Z 835.239,A -85,B 0,C 180,E1 15092.768,E2 15092.768} C_VEL
LIN {X 0,Y 481.383,Z 812.27,A -85,B 0,C 180,E1 15097.559,E2 15097.559} C_VEL
LIN {X 0,Y 470.794,Z 798.156,A -85,B 0,C 180,E1 15101.573,E2 15101.573} C_VEL
LIN {X 0,Y 465.769,Z 791.379,A -85,B 0,C 180,E1 15103.862,E2 15103.862} C_VEL
LIN {X 0,Y 461.764,Z 785.309,A -85,B 0,C 180,E1 15106.025,E2 15106.025} C_VEL
LIN {X 0,Y 456.764,Z 779.762,A -85,B 0,C 180,E1 15109.205,E2 15109.205} C_VEL
LIN {X 0,Y 455.588,Z 777.383,A -85,B 0,C 180,E1 15110.203,E2 15110.203} C_VEL
LIN {X 0,Y 450.687,Z 771.81,A -85,B 0,C 180,E1 15115.783,E2 15115.783} C_VEL
LIN {X 0,Y 450.245,Z 769.846,A -85,B 0,C 180,E1 15117.104,E2 15117.104} C_VEL
LIN {X 0,Y 450.547,Z 770.62,A -85,B 0,C 180,E1 15124.136,E2 15124.136} C_VEL
LIN {X 0,Y 453.651,Z 776.366,A -85,B 0,C 180,E1 15128.609,E2 15128.609} C_VEL
LIN {X 0,Y 456.27,Z 778.52,A -85,B 0,C 180,E1 15130.784,E2 15130.784} C_VEL
LIN {X 0,Y 459.769,Z 784.049,A -85,B 0,C 180,E1 15133.288,E2 15133.288} C_VEL
LIN {X 0,Y 461.953,Z 786.384,A -85,B 0,C 180,E1 15134.551,E2 15134.551} C_VEL
LIN {X 0,Y 467.961,Z 794.586,A -85,B 0,C 180,E1 15137.608,E2 15137.608} C_VEL
LIN {X 0,Y 473.463,Z 802.025,A -85,B 0,C 180,E1 15140.002,E2 15140.002} C_VEL
LIN {X 0,Y 483.182,Z 815.526,A -85,B 0,C 180,E1 15143.607,E2 15143.607} C_VEL
LIN {X 0,Y 496.748,Z 837.029,A -85,B 0,C 180,E1 15148.103,E2 15148.103} C_VEL
LIN {X 0,Y 510.886,Z 864.237,A -85,B 0,C 180,E1 15152.528,E2 15152.528} C_VEL
LIN {X 0,Y 523.643,Z 895.92,A -85,B 0,C 180,E1 15156.742,E2 15156.742} C_VEL
LIN {X 0,Y 513.522,Z 941.732,A -85,B 0,C 180,E1 15159.015,E2 15159.015} C_VEL
LIN {X 0,Y 502.051,Z 983.739,A -85,B 0,C 180,E1 15161.847,E2 15161.847} C_VEL
LIN {X 0,Y 489.29,Z 1024.394,A -85,B 0,C 180,E1 15165.471,E2 15165.471} C_VEL
LIN {X 0,Y 477.127,Z 1060.332,A -85,B 0,C 180,E1 15169.695,E2 15169.695} C_VEL
LIN {X 0,Y 465.619,Z 1093.774,A -85,B 0,C 180,E1 15174.828,E2 15174.828} C_VEL
LIN {X 0,Y 456.758,Z 1120.652,A -85,B 0,C 180,E1 15180.249,E2 15180.249} C_VEL
LIN {X 0,Y 450.113,Z 1143.324,A -85,B 0,C 180,E1 15186.244,E2 15186.244} C_VEL
LIN {X 0,Y 446.315,Z 1160.001,A -85,B 0,C 180,E1 15192.26,E2 15192.26} C_VEL
LIN {X 0,Y 444.466,Z 1171.445,A -85,B 0,C 180,E1 15198.231,E2 15198.231} C_VEL
LIN {X 0,Y 443.841,Z 1178.192,A -85,B 0,C 180,E1 15204.139,E2 15204.139} C_VEL
LIN {X 0,Y 443.888,Z 1180.444,A -85,B 0,C 180,E1 15210.001,E2 15210.001} C_VEL
LIN {X 0,Y 443.896,Z 1178.111,A -85,B 0,C 180,E1 15215.863,E2 15215.863} C_VEL
LIN {X 0,Y 444.359,Z 1172.819,A -85,B 0,C 180,E1 15220.781,E2 15220.781} C_VEL
LIN {X 0,Y 445.96,Z 1162.023,A -85,B 0,C 180,E1 15226.74,E2 15226.74} C_VEL
LIN {X 0,Y 449.788,Z 1144.935,A -85,B 0,C 180,E1 15233.175,E2 15233.175} C_VEL
LIN {X 0,Y 456.074,Z 1122.618,A -85,B 0,C 180,E1 15239.206,E2 15239.206} C_VEL
LIN {X 0,Y 465.323,Z 1094.728,A -85,B 0,C 180,E1 15244.916,E2 15244.916} C_VEL
LIN {X 0,Y 476.914,Z 1060.933,A -85,B 0,C 180,E1 15250.129,E2 15250.129} C_VEL
LIN {X 0,Y 488.971,Z 1025.547,A -85,B 0,C 180,E1 15254.312,E2 15254.312} C_VEL
LIN {X 0,Y 501.855,Z 984.253,A -85,B 0,C 180,E1 15258.019,E2 15258.019} C_VEL
LIN {X 0,Y 513.373,Z 942.04,A -85,B 0,C 180,E1 15260.88,E2 15260.88} C_VEL
LIN {X 0,Y 523.468,Z 895.231,A -85,B 0,C 180,E1 15263.234,E2 15263.234} C_VEL
LIN {X 0,Y 510.501,Z 863.529,A -85,B 0,C 180,E1 15267.477,E2 15267.477} C_VEL
LIN {X 0,Y 496.231,Z 836.265,A -85,B 0,C 180,E1 15271.939,E2 15271.939} C_VEL
LIN {X 0,Y 481.192,Z 812.439,A -85,B 0,C 180,E1 15276.967,E2 15276.967} C_VEL
LIN {X 0,Y 470.492,Z 798.037,A -85,B 0,C 180,E1 15281.097,E2 15281.097} C_VEL
LIN {X 0,Y 465.739,Z 791.543,A -85,B 0,C 180,E1 15283.278,E2 15283.278} C_VEL
LIN {X 0,Y 461.587,Z 785.405,A -85,B 0,C 180,E1 15285.497,E2 15285.497} C_VEL
LIN {X 0,Y 456.514,Z 779.476,A -85,B 0,C 180,E1 15288.739,E2 15288.739} C_VEL
LIN {X 0,Y 455.63,Z 777.417,A -85,B 0,C 180,E1 15289.502,E2 15289.502} C_VEL
LIN {X 0,Y 450.719,Z 772.03,A -85,B 0,C 180,E1 15294.782,E2 15294.782} C_VEL
LIN {X 0,Y 450.18,Z 769.822,A -85,B 0,C 180,E1 15296.162,E2 15296.162} C_VEL
LIN {X 0,Y 450.442,Z 770.521,A -85,B 0,C 180,E1 15303.978,E2 15303.978} C_VEL
LIN {X 0,Y 453.645,Z 776.387,A -85,B 0,C 180,E1 15308.39,E2 15308.39} C_VEL
LIN {X 0,Y 456.349,Z 778.445,A -85,B 0,C 180,E1 15310.564,E2 15310.564} C_VEL
LIN {X 0,Y 459.724,Z 783.883,A -85,B 0,C 180,E1 15312.949,E2 15312.949} C_VEL
LIN {X 0,Y 462.159,Z 786.277,A -85,B 0,C 180,E1 15314.325,E2 15314.325} C_VEL
LIN {X 0,Y 466.858,Z 792.113,A -85,B 0,C 180,E1 15316.703,E2 15316.703} C_VEL
LIN {X 0,Y 478.348,Z 808.124,A -85,B 0,C 180,E1 15321.409,E2 15321.409} C_VEL
LIN {X 0,Y 491.363,Z 827.011,A -85,B 0,C 180,E1 15325.692,E2 15325.692} C_VEL
LIN {X 0,Y 507.029,Z 853.129,A -85,B 0,C 180,E1 15330.271,E2 15330.271} C_VEL
LIN {X 0,Y 522.707,Z 885.469,A -85,B 0,C 180,E1 15334.698,E2 15334.698} C_VEL
LIN {X 0,Y 526.458,Z 896.483,A -85,B 0,C 180,E1 15335.914,E2 15335.914} C_VEL
LIN {X 0,Y 516.69,Z 944.806,A -85,B 0,C 180,E1 15337.938,E2 15337.938} C_VEL
LIN {X 0,Y 505.343,Z 989.525,A -85,B 0,C 180,E1 15340.574,E2 15340.574} C_VEL
LIN {X 0,Y 492.899,Z 1032.247,A -85,B 0,C 180,E1 15343.953,E2 15343.953} C_VEL
LIN {X 0,Y 480.883,Z 1069.691,A -85,B 0,C 180,E1 15347.838,E2 15347.838} C_VEL
LIN {X 0,Y 468.794,Z 1106.539,A -85,B 0,C 180,E1 15352.815,E2 15352.815} C_VEL
LIN {X 0,Y 458.946,Z 1137.031,A -85,B 0,C 180,E1 15358.209,E2 15358.209} C_VEL
LIN {X 0,Y 451.613,Z 1163.104,A -85,B 0,C 180,E1 15364.215,E2 15364.215} C_VEL
LIN {X 0,Y 447.161,Z 1182.521,A -85,B 0,C 180,E1 15370.248,E2 15370.248} C_VEL
LIN {X 0,Y 444.853,Z 1196.476,A -85,B 0,C 180,E1 15376.243,E2 15376.243} C_VEL
LIN {X 0,Y 444.053,Z 1205.363,A -85,B 0,C 180,E1 15382.176,E2 15382.176} C_VEL
LIN {X 0,Y 443.853,Z 1209.241,A -85,B 0,C 180,E1 15388.048,E2 15388.048} C_VEL
LIN {X 0,Y 444.048,Z 1209.248,A -85,B 0,C 180,E1 15391.949,E2 15391.949} C_VEL
LIN {X 0,Y 444.056,Z 1205.367,A -85,B 0,C 180,E1 15397.822,E2 15397.822} C_VEL
LIN {X 0,Y 444.052,Z 1204.723,A -85,B 0,C 180,E1 15398.337,E2 15398.337} C_VEL
LIN {X 0,Y 440.273,Z 1201.963,A -85,B 0,C 180,E1 15400.522,E2 15400.522} C_VEL
LIN {X 0,Y 436.686,Z 1198.48,A -85,B 0,C 180,E1 15402.736,E2 15402.736} C_VEL
LIN {X 0,Y 438.64,Z 1186.476,A -85,B 0,C 180,E1 15408.529,E2 15408.529} C_VEL
LIN {X 0,Y 442.934,Z 1167.536,A -85,B 0,C 180,E1 15414.894,E2 15414.894} C_VEL
LIN {X 0,Y 450.133,Z 1142.689,A -85,B 0,C 180,E1 15421.118,E2 15421.118} C_VEL
LIN {X 0,Y 460.111,Z 1112.311,A -85,B 0,C 180,E1 15426.824,E2 15426.824} C_VEL
LIN {X 0,Y 471.7,Z 1078.475,A -85,B 0,C 180,E1 15431.733,E2 15431.733} C_VEL
LIN {X 0,Y 485.208,Z 1038.055,A -85,B 0,C 180,E1 15436.183,E2 15436.183} C_VEL
LIN {X 0,Y 497.999,Z 996.597,A -85,B 0,C 180,E1 15439.629,E2 15439.629} C_VEL
LIN {X 0,Y 510.697,Z 949.365,A -85,B 0,C 180,E1 15442.526,E2 15442.526} C_VEL
LIN {X 0,Y 520.121,Z 906.135,A -85,B 0,C 180,E1 15444.436,E2 15444.436} C_VEL
LIN {X 0,Y 521.186,Z 898.596,A -85,B 0,C 180,E1 15444.752,E2 15444.752} C_VEL
LIN {X 0,Y 507.538,Z 867.446,A -85,B 0,C 180,E1 15448.903,E2 15448.903} C_VEL
LIN {X 0,Y 493.021,Z 841.188,A -85,B 0,C 180,E1 15453.253,E2 15453.253} C_VEL
LIN {X 0,Y 478.857,Z 819.092,A -85,B 0,C 180,E1 15457.977,E2 15457.977} C_VEL
LIN {X 0,Y 468.776,Z 805.216,A -85,B 0,C 180,E1 15461.977,E2 15461.977} C_VEL
LIN {X 0,Y 464.34,Z 799.008,A -85,B 0,C 180,E1 15464.054,E2 15464.054} C_VEL
LIN {X 0,Y 459.158,Z 792.106,A -85,B 0,C 180,E1 15466.913,E2 15466.913} C_VEL
LIN {X 0,Y 455.161,Z 786.481,A -85,B 0,C 180,E1 15469.711,E2 15469.711} C_VEL
LIN {X 0,Y 453.449,Z 784.701,A -85,B 0,C 180,E1 15471.124,E2 15471.124} C_VEL
LIN {X 0,Y 449.503,Z 778.698,A -85,B 0,C 180,E1 15476.375,E2 15476.375} C_VEL
LIN {X 0,Y 448.95,Z 777.582,A -85,B 0,C 180,E1 15478.06,E2 15478.06} C_VEL
LIN {X 0,Y 449.519,Z 778.499,A -85,B 0,C 180,E1 15484.024,E2 15484.024} C_VEL
LIN {X 0,Y 452.954,Z 784.416,A -85,B 0,C 180,E1 15488.864,E2 15488.864} C_VEL
LIN {X 0,Y 454.988,Z 786.3,A -85,B 0,C 180,E1 15490.573,E2 15490.573} C_VEL
LIN {X 0,Y 458.824,Z 791.955,A -85,B 0,C 180,E1 15493.316,E2 15493.316} C_VEL
LIN {X 0,Y 460.842,Z 794.752,A -85,B 0,C 180,E1 15494.527,E2 15494.527} C_VEL
LIN {X 0,Y 466.256,Z 802.098,A -85,B 0,C 180,E1 15497.37,E2 15497.37} C_VEL
LIN {X 0,Y 472.104,Z 810.231,A -85,B 0,C 180,E1 15499.973,E2 15499.973} C_VEL
LIN {X 0,Y 483.197,Z 826.186,A -85,B 0,C 180,E1 15504.219,E2 15504.219} C_VEL
LIN {X 0,Y 497.09,Z 850.335,A -85,B 0,C 180,E1 15508.958,E2 15508.958} C_VEL
LIN {X 0,Y 509.868,Z 877.379,A -85,B 0,C 180,E1 15513.21,E2 15513.21} C_VEL
LIN {X 0,Y 518.188,Z 899.573,A -85,B 0,C 180,E1 15516.177,E2 15516.177} C_VEL
LIN {X 0,Y 507.84,Z 944.756,A -85,B 0,C 180,E1 15518.472,E2 15518.472} C_VEL
LIN {X 0,Y 495.702,Z 987.124,A -85,B 0,C 180,E1 15521.398,E2 15521.398} C_VEL
LIN {X 0,Y 482.852,Z 1026.716,A -85,B 0,C 180,E1 15525.003,E2 15525.003} C_VEL
LIN {X 0,Y 470.111,Z 1062.792,A -85,B 0,C 180,E1 15529.353,E2 15529.353} C_VEL
LIN {X 0,Y 458.426,Z 1095.467,A -85,B 0,C 180,E1 15534.482,E2 15534.482} C_VEL
LIN {X 0,Y 449.001,Z 1122.85,A -85,B 0,C 180,E1 15540.188,E2 15540.188} C_VEL
LIN {X 0,Y 442.213,Z 1145.173,A -85,B 0,C 180,E1 15546.301,E2 15546.301} C_VEL
LIN {X 0,Y 438.383,Z 1161.378,A -85,B 0,C 180,E1 15552.446,E2 15552.446} C_VEL
LIN {X 0,Y 436.617,Z 1171.707,A -85,B 0,C 180,E1 15558.016,E2 15558.016} C_VEL
LIN {X 0,Y 435.955,Z 1178.452,A -85,B 0,C 180,E1 15564.032,E2 15564.032} C_VEL
LIN {X 0,Y 435.991,Z 1180.704,A -85,B 0,C 180,E1 15570.001,E2 15570.001} C_VEL
LIN {X 0,Y 436.006,Z 1178.372,A -85,B 0,C 180,E1 15575.969,E2 15575.969} C_VEL
LIN {X 0,Y 436.499,Z 1173.083,A -85,B 0,C 180,E1 15580.977,E2 15580.977} C_VEL
LIN {X 0,Y 438.238,Z 1162.29,A -85,B 0,C 180,E1 15587.044,E2 15587.044} C_VEL
LIN {X 0,Y 441.998,Z 1146.224,A -85,B 0,C 180,E1 15593.244,E2 15593.244} C_VEL
LIN {X 0,Y 448.465,Z 1124.309,A -85,B 0,C 180,E1 15599.38,E2 15599.38} C_VEL
LIN {X 0,Y 458.109,Z 1096.352,A -85,B 0,C 180,E1 15605.259,E2 15605.259} C_VEL
LIN {X 0,Y 469.692,Z 1063.918,A -85,B 0,C 180,E1 15610.398,E2 15610.398} C_VEL
LIN {X 0,Y 482.748,Z 1027.143,A -85,B 0,C 180,E1 15614.853,E2 15614.853} C_VEL
LIN {X 0,Y 495.61,Z 987.272,A -85,B 0,C 180,E1 15618.497,E2 15618.497} C_VEL
LIN {X 0,Y 507.775,Z 944.641,A -85,B 0,C 180,E1 15621.45,E2 15621.45} C_VEL
LIN {X 0,Y 517.798,Z 902.137,A -85,B 0,C 180,E1 15623.593,E2 15623.593} C_VEL
LIN {X 0,Y 518.008,Z 898.779,A -85,B 0,C 180,E1 15623.809,E2 15623.809} C_VEL
LIN {X 0,Y 505.304,Z 866.86,A -85,B 0,C 180,E1 15628.224,E2 15628.224} C_VEL
LIN {X 0,Y 492.171,Z 841.703,A -85,B 0,C 180,E1 15632.522,E2 15632.522} C_VEL
LIN {X 0,Y 478.63,Z 819.386,A -85,B 0,C 180,E1 15637.321,E2 15637.321} C_VEL
LIN {X 0,Y 468.41,Z 805.205,A -85,B 0,C 180,E1 15641.456,E2 15641.456} C_VEL
LIN {X 0,Y 463.759,Z 798.75,A -85,B 0,C 180,E1 15643.706,E2 15643.706} C_VEL
LIN {X 0,Y 458.889,Z 792.007,A -85,B 0,C 180,E1 15646.444,E2 15646.444} C_VEL
LIN {X 0,Y 454.912,Z 786.188,A -85,B 0,C 180,E1 15649.244,E2 15649.244} C_VEL
LIN {X 0,Y 449.485,Z 778.976,A -85,B 0,C 180,E1 15655.372,E2 15655.372} C_VEL
LIN {X 0,Y 448.822,Z 777.565,A -85,B 0,C 180,E1 15657.117,E2 15657.117} C_VEL
LIN {X 0,Y 449.401,Z 778.459,A -85,B 0,C 180,E1 15663.867,E2 15663.867} C_VEL
LIN {X 0,Y 452.956,Z 784.436,A -85,B 0,C 180,E1 15668.644,E2 15668.644} C_VEL
LIN {X 0,Y 455.054,Z 786.264,A -85,B 0,C 180,E1 15670.352,E2 15670.352} C_VEL
LIN {X 0,Y 458.974,Z 791.964,A -85,B 0,C 180,E1 15673.092,E2 15673.092} C_VEL
LIN {X 0,Y 460.94,Z 794.526,A -85,B 0,C 180,E1 15674.243,E2 15674.243} C_VEL
LIN {X 0,Y 466.535,Z 801.973,A -85,B 0,C 180,E1 15677.079,E2 15677.079} C_VEL
LIN {X 0,Y 475.832,Z 814.624,A -85,B 0,C 180,E1 15680.952,E2 15680.952} C_VEL
LIN {X 0,Y 488.885,Z 834.36,A -85,B 0,C 180,E1 15685.465,E2 15685.465} C_VEL
LIN {X 0,Y 503.801,Z 860.22,A -85,B 0,C 180,E1 15690.031,E2 15690.031} C_VEL
LIN {X 0,Y 518.571,Z 891.833,A -85,B 0,C 180,E1 15694.422,E2 15694.422} C_VEL
LIN {X 0,Y 521.163,Z 898.421,A -85,B 0,C 180,E1 15695.245,E2 15695.245} C_VEL
LIN {X 0,Y 511.24,Z 946.842,A -85,B 0,C 180,E1 15697.336,E2 15697.336} C_VEL
LIN {X 0,Y 499.143,Z 992.454,A -85,B 0,C 180,E1 15700.086,E2 15700.086} C_VEL
LIN {X 0,Y 486.343,Z 1034.791,A -85,B 0,C 180,E1 15703.511,E2 15703.511} C_VEL
LIN {X 0,Y 474.029,Z 1071.553,A -85,B 0,C 180,E1 15707.426,E2 15707.426} C_VEL
LIN {X 0,Y 461.64,Z 1107.843,A -85,B 0,C 180,E1 15712.434,E2 15712.434} C_VEL
LIN {X 0,Y 451.162,Z 1139.104,A -85,B 0,C 180,E1 15718.137,E2 15718.137} C_VEL
LIN {X 0,Y 443.848,Z 1164.014,A -85,B 0,C 180,E1 15724.088,E2 15724.088} C_VEL
LIN {X 0,Y 439.142,Z 1183.757,A -85,B 0,C 180,E1 15730.448,E2 15730.448} C_VEL
LIN {X 0,Y 437.027,Z 1196.212,A -85,B 0,C 180,E1 15735.992,E2 15735.992} C_VEL
LIN {X 0,Y 436.163,Z 1205.102,A -85,B 0,C 180,E1 15742.033,E2 15742.033} C_VEL
LIN {X 0,Y 435.97,Z 1208.982,A -85,B 0,C 180,E1 15748.013,E2 15748.013} C_VEL
LIN {X 0,Y 436.141,Z 1208.988,A -85,B 0,C 180,E1 15751.985,E2 15751.985} C_VEL
LIN {X 0,Y 436.163,Z 1204.648,A -85,B 0,C 180,E1 15758.338,E2 15758.338} C_VEL
LIN {X 0,Y 436.686,Z 1198.48,A -85,B 0,C 180,E1 15762.736,E2 15762.736} C_VEL
LIN {X 0,Y 433.373,Z 1194.65,A -85,B 0,C 180,E1 15764.945,E2 15764.945} C_VEL
LIN {X 0,Y 430.143,Z 1190.084,A -85,B 0,C 180,E1 15767.166,E2 15767.166} C_VEL
LIN {X 0,Y 433.866,Z 1172.994,A -85,B 0,C 180,E1 15773.61,E2 15773.61} C_VEL
LIN {X 0,Y 440.123,Z 1151.474,A -85,B 0,C 180,E1 15779.573,E2 15779.573} C_VEL
LIN {X 0,Y 449.945,Z 1121.884,A -85,B 0,C 180,E1 15785.76,E2 15785.76} C_VEL
LIN {X 0,Y 461.489,Z 1089.411,A -85,B 0,C 180,E1 15790.91,E2 15790.91} C_VEL
LIN {X 0,Y 474.995,Z 1051.064,A -85,B 0,C 180,E1 15795.574,E2 15795.574} C_VEL
LIN {X 0,Y 488.573,Z 1010.083,A -85,B 0,C 180,E1 15799.301,E2 15799.301} C_VEL
LIN {X 0,Y 501.161,Z 967.32,A -85,B 0,C 180,E1 15802.235,E2 15802.235} C_VEL
LIN {X 0,Y 512.067,Z 921.751,A -85,B 0,C 180,E1 15804.545,E2 15804.545} C_VEL
LIN {X 0,Y 515.738,Z 901.948,A -85,B 0,C 180,E1 15805.379,E2 15805.379} C_VEL
LIN {X 0,Y 502.537,Z 871.111,A -85,B 0,C 180,E1 15809.625,E2 15809.625} C_VEL
LIN {X 0,Y 487.464,Z 843.499,A -85,B 0,C 180,E1 15814.44,E2 15814.44} C_VEL
LIN {X 0,Y 475.553,Z 824.878,A -85,B 0,C 180,E1 15818.691,E2 15818.691} C_VEL
LIN {X 0,Y 466.521,Z 812.064,A -85,B 0,C 180,E1 15822.435,E2 15822.435} C_VEL
LIN {X 0,Y 462.403,Z 806.24,A -85,B 0,C 180,E1 15824.48,E2 15824.48} C_VEL
LIN {X 0,Y 457.813,Z 799.742,A -85,B 0,C 180,E1 15827.117,E2 15827.117} C_VEL
LIN {X 0,Y 453.825,Z 794.018,A -85,B 0,C 180,E1 15829.983,E2 15829.983} C_VEL
LIN {X 0,Y 448.448,Z 786.312,A -85,B 0,C 180,E1 15836.609,E2 15836.609} C_VEL
LIN {X 0,Y 448.429,Z 785.698,A -85,B 0,C 180,E1 15843.611,E2 15843.611} C_VEL
LIN {X 0,Y 451.244,Z 791.751,A -85,B 0,C 180,E1 15848.17,E2 15848.17} C_VEL
LIN {X 0,Y 453.723,Z 793.995,A -85,B 0,C 180,E1 15850.36,E2 15850.36} C_VEL
LIN {X 0,Y 457.827,Z 799.87,A -85,B 0,C 180,E1 15853.345,E2 15853.345} C_VEL
LIN {X 0,Y 464.742,Z 809.983,A -85,B 0,C 180,E1 15857.246,E2 15857.246} C_VEL
LIN {X 0,Y 473.097,Z 821.694,A -85,B 0,C 180,E1 15860.991,E2 15860.991} C_VEL
LIN {X 0,Y 485.138,Z 841.282,A -85,B 0,C 180,E1 15865.647,E2 15865.647} C_VEL
LIN {X 0,Y 498.411,Z 866.635,A -85,B 0,C 180,E1 15870.315,E2 15870.315} C_VEL
LIN {X 0,Y 510.818,Z 897.291,A -85,B 0,C 180,E1 15874.822,E2 15874.822} C_VEL
LIN {X 0,Y 512.733,Z 904.211,A -85,B 0,C 180,E1 15875.665,E2 15875.665} C_VEL
LIN {X 0,Y 502.562,Z 946.174,A -85,B 0,C 180,E1 15877.828,E2 15877.828} C_VEL
LIN {X 0,Y 490.112,Z 988.271,A -85,B 0,C 180,E1 15880.76,E2 15880.76} C_VEL
LIN {X 0,Y 476.495,Z 1028.754,A -85,B 0,C 180,E1 15884.498,E2 15884.498} C_VEL
LIN {X 0,Y 463.124,Z 1065.224,A -85,B 0,C 180,E1 15888.997,E2 15888.997} C_VEL
LIN {X 0,Y 451.253,Z 1097.047,A -85,B 0,C 180,E1 15894.126,E2 15894.126} C_VEL
LIN {X 0,Y 441.106,Z 1125.43,A -85,B 0,C 180,E1 15900.217,E2 15900.217} C_VEL
LIN {X 0,Y 434.237,Z 1147.008,A -85,B 0,C 180,E1 15906.411,E2 15906.411} C_VEL
LIN {X 0,Y 430.419,Z 1162.756,A -85,B 0,C 180,E1 15912.638,E2 15912.638} C_VEL
LIN {X 0,Y 428.614,Z 1173.484,A -85,B 0,C 180,E1 15918.82,E2 15918.82} C_VEL
LIN {X 0,Y 428.061,Z 1178.712,A -85,B 0,C 180,E1 15923.922,E2 15923.922} C_VEL
LIN {X 0,Y 428.093,Z 1180.963,A -85,B 0,C 180,E1 15930.001,E2 15930.001} C_VEL
LIN {X 0,Y 428.112,Z 1178.633,A -85,B 0,C 180,E1 15936.08,E2 15936.08} C_VEL
LIN {X 0,Y 428.667,Z 1173.346,A -85,B 0,C 180,E1 15941.18,E2 15941.18} C_VEL
LIN {X 0,Y 430.503,Z 1162.557,A -85,B 0,C 180,E1 15947.36,E2 15947.36} C_VEL
LIN {X 0,Y 434.42,Z 1146.749,A -85,B 0,C 180,E1 15953.581,E2 15953.581} C_VEL
LIN {X 0,Y 441.153,Z 1125.085,A -85,B 0,C 180,E1 15959.782,E2 15959.782} C_VEL
LIN {X 0,Y 451.414,Z 1096.625,A -85,B 0,C 180,E1 15965.862,E2 15965.862} C_VEL
LIN {X 0,Y 463.365,Z 1064.51,A -85,B 0,C 180,E1 15971.01,E2 15971.01} C_VEL
LIN {X 0,Y 476.609,Z 1028.552,A -85,B 0,C 180,E1 15975.421,E2 15975.421} C_VEL
LIN {X 0,Y 489.853,Z 988.916,A -85,B 0,C 180,E1 15979.095,E2 15979.095} C_VEL
LIN {X 0,Y 502.971,Z 944.29,A -85,B 0,C 180,E1 15982.201,E2 15982.201} C_VEL
LIN {X 0,Y 512.854,Z 903.142,A -85,B 0,C 180,E1 15984.294,E2 15984.294} C_VEL
LIN {X 0,Y 501.471,Z 873.31,A -85,B 0,C 180,E1 15988.518,E2 15988.518} C_VEL
LIN {X 0,Y 488.591,Z 847.688,A -85,B 0,C 180,E1 15992.979,E2 15992.979} C_VEL
LIN {X 0,Y 475.833,Z 826.131,A -85,B 0,C 180,E1 15997.735,E2 15997.735} C_VEL
LIN {X 0,Y 466.534,Z 812.525,A -85,B 0,C 180,E1 16001.739,E2 16001.739} C_VEL
LIN {X 0,Y 461.937,Z 806.125,A -85,B 0,C 180,E1 16004.013,E2 16004.013} C_VEL
LIN {X 0,Y 457.497,Z 799.664,A -85,B 0,C 180,E1 16006.645,E2 16006.645} C_VEL
LIN {X 0,Y 453.582,Z 793.683,A -85,B 0,C 180,E1 16009.515,E2 16009.515} C_VEL
LIN {X 0,Y 448.413,Z 786.594,A -85,B 0,C 180,E1 16015.603,E2 16015.603} C_VEL
LIN {X 0,Y 447.86,Z 785.406,A -85,B 0,C 180,E1 16017.111,E2 16017.111} C_VEL
LIN {X 0,Y 448.367,Z 786.347,A -85,B 0,C 180,E1 16023.755,E2 16023.755} C_VEL
LIN {X 0,Y 452.279,Z 792.456,A -85,B 0,C 180,E1 16028.899,E2 16028.899} C_VEL
LIN {X 0,Y 453.904,Z 794.346,A -85,B 0,C 180,E1 16030.257,E2 16030.257} C_VEL
LIN {X 0,Y 458.439,Z 800.122,A -85,B 0,C 180,E1 16033.35,E2 16033.35} C_VEL
LIN {X 0,Y 465.319,Z 810.244,A -85,B 0,C 180,E1 16037.064,E2 16037.064} C_VEL
LIN {X 0,Y 473.928,Z 822.204,A -85,B 0,C 180,E1 16040.728,E2 16040.728} C_VEL
LIN {X 0,Y 486.22,Z 841.441,A -85,B 0,C 180,E1 16045.183,E2 16045.183} C_VEL
LIN {X 0,Y 500.506,Z 867.084,A -85,B 0,C 180,E1 16049.761,E2 16049.761} C_VEL
LIN {X 0,Y 514.396,Z 898.401,A -85,B 0,C 180,E1 16054.189,E2 16054.189} C_VEL
LIN {X 0,Y 515.922,Z 902.831,A -85,B 0,C 180,E1 16054.72,E2 16054.72} C_VEL
LIN {X 0,Y 505.82,Z 948.733,A -85,B 0,C 180,E1 16056.724,E2 16056.724} C_VEL
LIN {X 0,Y 492.987,Z 995.413,A -85,B 0,C 180,E1 16059.589,E2 16059.589} C_VEL
LIN {X 0,Y 479.895,Z 1036.842,A -85,B 0,C 180,E1 16063.025,E2 16063.025} C_VEL
LIN {X 0,Y 466.727,Z 1074.733,A -85,B 0,C 180,E1 16067.162,E2 16067.162} C_VEL
LIN {X 0,Y 454.493,Z 1109.047,A -85,B 0,C 180,E1 16072.04,E2 16072.04} C_VEL
LIN {X 0,Y 443.586,Z 1140.472,A -85,B 0,C 180,E1 16077.914,E2 16077.914} C_VEL
LIN {X 0,Y 436.124,Z 1164.76,A -85,B 0,C 180,E1 16083.911,E2 16083.911} C_VEL
LIN {X 0,Y 431.248,Z 1184.477,A -85,B 0,C 180,E1 16090.46,E2 16090.46} C_VEL
LIN {X 0,Y 429.223,Z 1195.948,A -85,B 0,C 180,E1 16095.732,E2 16095.732} C_VEL
LIN {X 0,Y 428.262,Z 1204.84,A -85,B 0,C 180,E1 16101.885,E2 16101.885} C_VEL
LIN {X 0,Y 428.069,Z 1208.722,A -85,B 0,C 180,E1 16107.976,E2 16107.976} C_VEL
LIN {X 0,Y 428.236,Z 1208.729,A -85,B 0,C 180,E1 16112.021,E2 16112.021} C_VEL
LIN {X 0,Y 428.264,Z 1204.843,A -85,B 0,C 180,E1 16118.113,E2 16118.113} C_VEL
LIN {X 0,Y 429.205,Z 1195.95,A -85,B 0,C 180,E1 16124.267,E2 16124.267} C_VEL
LIN {X 0,Y 430.143,Z 1190.084,A -85,B 0,C 180,E1 16127.166,E2 16127.166} C_VEL
LIN {X 0,Y 427.193,Z 1185.244,A -85,B 0,C 180,E1 16129.38,E2 16129.38} C_VEL
LIN {X 0,Y 424.527,Z 1179.817,A -85,B 0,C 180,E1 16131.61,E2 16131.61} C_VEL
LIN {X 0,Y 429.749,Z 1160.829,A -85,B 0,C 180,E1 16137.619,E2 16137.619} C_VEL
LIN {X 0,Y 438.659,Z 1134.166,A -85,B 0,C 180,E1 16143.945,E2 16143.945} C_VEL
LIN {X 0,Y 449.711,Z 1104.02,A -85,B 0,C 180,E1 16149.381,E2 16149.381} C_VEL
LIN {X 0,Y 463.261,Z 1067.455,A -85,B 0,C 180,E1 16154.411,E2 16154.411} C_VEL
LIN {X 0,Y 476.399,Z 1030.515,A -85,B 0,C 180,E1 16158.277,E2 16158.277} C_VEL
LIN {X 0,Y 490.276,Z 987.253,A -85,B 0,C 180,E1 16161.706,E2 16161.706} C_VEL
LIN {X 0,Y 502.419,Z 943.011,A -85,B 0,C 180,E1 16164.297,E2 16164.297} C_VEL
LIN {X 0,Y 510.506,Z 905.599,A -85,B 0,C 180,E1 16165.975,E2 16165.975} C_VEL
LIN {X 0,Y 497.659,Z 875.267,A -85,B 0,C 180,E1 16170.302,E2 16170.302} C_VEL
LIN {X 0,Y 484.096,Z 849.598,A -85,B 0,C 180,E1 16174.92,E2 16174.92} C_VEL
LIN {X 0,Y 472.925,Z 831.623,A -85,B 0,C 180,E1 16179.095,E2 16179.095} C_VEL
LIN {X 0,Y 464.518,Z 819.257,A -85,B 0,C 180,E1 16182.784,E2 16182.784} C_VEL
LIN {X 0,Y 460.515,Z 813.477,A -85,B 0,C 180,E1 16184.833,E2 16184.833} C_VEL
LIN {X 0,Y 456.075,Z 807.12,A -85,B 0,C 180,E1 16187.524,E2 16187.524} C_VEL
LIN {X 0,Y 452.332,Z 800.941,A -85,B 0,C 180,E1 16190.435,E2 16190.435} C_VEL
LIN {X 0,Y 447.466,Z 794.563,A -85,B 0,C 180,E1 16196.541,E2 16196.541} C_VEL
LIN {X 0,Y 447.026,Z 793.264,A -85,B 0,C 180,E1 16198.052,E2 16198.052} C_VEL
LIN {X 0,Y 447.454,Z 794.114,A -85,B 0,C 180,E1 16203.74,E2 16203.74} C_VEL
LIN {X 0,Y 451.016,Z 800.131,A -85,B 0,C 180,E1 16208.902,E2 16208.902} C_VEL
LIN {X 0,Y 452.531,Z 802.155,A -85,B 0,C 180,E1 16210.299,E2 16210.299} C_VEL
LIN {X 0,Y 457.733,Z 809.971,A -85,B 0,C 180,E1 16214.088,E2 16214.088} C_VEL
LIN {X 0,Y 463.384,Z 818.158,A -85,B 0,C 180,E1 16217.237,E2 16217.237} C_VEL
LIN {X 0,Y 470.832,Z 829.05,A -85,B 0,C 180,E1 16220.747,E2 16220.747} C_VEL
LIN {X 0,Y 482.634,Z 849.023,A -85,B 0,C 180,E1 16225.532,E2 16225.532} C_VEL
LIN {X 0,Y 495.029,Z 873.978,A -85,B 0,C 180,E1 16230.147,E2 16230.147} C_VEL
LIN {X 0,Y 506.274,Z 903.274,A -85,B 0,C 180,E1 16234.532,E2 16234.532} C_VEL
LIN {X 0,Y 507.521,Z 907.234,A -85,B 0,C 180,E1 16235.051,E2 16235.051} C_VEL
LIN {X 0,Y 496.497,Z 950.478,A -85,B 0,C 180,E1 16237.35,E2 16237.35} C_VEL
LIN {X 0,Y 483.406,Z 993.043,A -85,B 0,C 180,E1 16240.4,E2 16240.4} C_VEL
LIN {X 0,Y 470.138,Z 1030.788,A -85,B 0,C 180,E1 16243.988,E2 16243.988} C_VEL
LIN {X 0,Y 455.793,Z 1068.627,A -85,B 0,C 180,E1 16248.769,E2 16248.769} C_VEL
LIN {X 0,Y 443.546,Z 1100.099,A -85,B 0,C 180,E1 16254.052,E2 16254.052} C_VEL
LIN {X 0,Y 433.283,Z 1127.818,A -85,B 0,C 180,E1 16260.201,E2 16260.201} C_VEL
LIN {X 0,Y 426.289,Z 1148.767,A -85,B 0,C 180,E1 16266.499,E2 16266.499} C_VEL
LIN {X 0,Y 422.469,Z 1164.134,A -85,B 0,C 180,E1 16272.838,E2 16272.838} C_VEL
LIN {X 0,Y 420.782,Z 1173.745,A -85,B 0,C 180,E1 16278.609,E2 16278.609} C_VEL
LIN {X 0,Y 420.181,Z 1178.971,A -85,B 0,C 180,E1 16283.807,E2 16283.807} C_VEL
LIN {X 0,Y 420.214,Z 1181.222,A -85,B 0,C 180,E1 16290.001,E2 16290.001} C_VEL
LIN {X 0,Y 420.232,Z 1178.894,A -85,B 0,C 180,E1 16296.194,E2 16296.194} C_VEL
LIN {X 0,Y 420.831,Z 1173.609,A -85,B 0,C 180,E1 16301.391,E2 16301.391} C_VEL
LIN {X 0,Y 422.778,Z 1162.825,A -85,B 0,C 180,E1 16307.688,E2 16307.688} C_VEL
LIN {X 0,Y 426.905,Z 1147.021,A -85,B 0,C 180,E1 16314.022,E2 16314.022} C_VEL
LIN {X 0,Y 434.005,Z 1125.358,A -85,B 0,C 180,E1 16320.323,E2 16320.323} C_VEL
LIN {X 0,Y 444.654,Z 1097.1,A -85,B 0,C 180,E1 16326.447,E2 16326.447} C_VEL
LIN {X 0,Y 457.058,Z 1065.136,A -85,B 0,C 180,E1 16331.636,E2 16331.636} C_VEL
LIN {X 0,Y 470.655,Z 1029.55,A -85,B 0,C 180,E1 16336.045,E2 16336.045} C_VEL
LIN {X 0,Y 484.238,Z 990.294,A -85,B 0,C 180,E1 16339.728,E2 16339.728} C_VEL
LIN {X 0,Y 497.703,Z 945.992,A -85,B 0,C 180,E1 16342.844,E2 16342.844} C_VEL
LIN {X 0,Y 507.576,Z 906.981,A -85,B 0,C 180,E1 16344.856,E2 16344.856} C_VEL
LIN {X 0,Y 496.269,Z 876.777,A -85,B 0,C 180,E1 16349.269,E2 16349.269} C_VEL
LIN {X 0,Y 483.268,Z 850.279,A -85,B 0,C 180,E1 16354.099,E2 16354.099} C_VEL
LIN {X 0,Y 471.96,Z 831.237,A -85,B 0,C 180,E1 16358.602,E2 16358.602} C_VEL
LIN {X 0,Y 464.033,Z 819.203,A -85,B 0,C 180,E1 16362.252,E2 16362.252} C_VEL
LIN {X 0,Y 459.973,Z 813.269,A -85,B 0,C 180,E1 16364.408,E2 16364.408} C_VEL
LIN {X 0,Y 455.809,Z 807.142,A -85,B 0,C 180,E1 16366.956,E2 16366.956} C_VEL
LIN {X 0,Y 451.291,Z 800.279,A -85,B 0,C 180,E1 16370.576,E2 16370.576} C_VEL
LIN {X 0,Y 447.388,Z 794.414,A -85,B 0,C 180,E1 16375.714,E2 16375.714} C_VEL
LIN {X 0,Y 446.626,Z 793.149,A -85,B 0,C 180,E1 16378.073,E2 16378.073} C_VEL
LIN {X 0,Y 447.341,Z 794.189,A -85,B 0,C 180,E1 16383.642,E2 16383.642} C_VEL
LIN {X 0,Y 451.326,Z 800.31,A -85,B 0,C 180,E1 16388.918,E2 16388.918} C_VEL
LIN {X 0,Y 452.76,Z 802.396,A -85,B 0,C 180,E1 16390.162,E2 16390.162} C_VEL
LIN {X 0,Y 457.974,Z 809.686,A -85,B 0,C 180,E1 16393.789,E2 16393.789} C_VEL
LIN {X 0,Y 463.851,Z 818.184,A -85,B 0,C 180,E1 16396.963,E2 16396.963} C_VEL
LIN {X 0,Y 472.288,Z 830.39,A -85,B 0,C 180,E1 16400.678,E2 16400.678} C_VEL
LIN {X 0,Y 485.029,Z 850.908,A -85,B 0,C 180,E1 16405.429,E2 16405.429} C_VEL
LIN {X 0,Y 499.011,Z 878.152,A -85,B 0,C 180,E1 16410.173,E2 16410.173} C_VEL
LIN {X 0,Y 510.66,Z 905.988,A -85,B 0,C 180,E1 16414.09,E2 16414.09} C_VEL
LIN {X 0,Y 500.124,Z 951.76,A -85,B 0,C 180,E1 16416.157,E2 16416.157} C_VEL
LIN {X 0,Y 486.781,Z 998.625,A -85,B 0,C 180,E1 16419.096,E2 16419.096} C_VEL
LIN {X 0,Y 472.861,Z 1040.589,A -85,B 0,C 180,E1 16422.691,E2 16422.691} C_VEL
LIN {X 0,Y 459.3,Z 1078.343,A -85,B 0,C 180,E1 16426.945,E2 16426.945} C_VEL
LIN {X 0,Y 446.685,Z 1112.104,A -85,B 0,C 180,E1 16431.95,E2 16431.95} C_VEL
LIN {X 0,Y 436.044,Z 1141.7,A -85,B 0,C 180,E1 16437.653,E2 16437.653} C_VEL
LIN {X 0,Y 428.186,Z 1166.212,A -85,B 0,C 180,E1 16443.938,E2 16443.938} C_VEL
LIN {X 0,Y 423.478,Z 1184.452,A -85,B 0,C 180,E1 16450.183,E2 16450.183} C_VEL
LIN {X 0,Y 421.107,Z 1197.589,A -85,B 0,C 180,E1 16456.546,E2 16456.546} C_VEL
LIN {X 0,Y 420.365,Z 1204.578,A -85,B 0,C 180,E1 16461.732,E2 16461.732} C_VEL
LIN {X 0,Y 420.197,Z 1208.464,A -85,B 0,C 180,E1 16467.938,E2 16467.938} C_VEL
LIN {X 0,Y 420.346,Z 1208.469,A -85,B 0,C 180,E1 16472.059,E2 16472.059} C_VEL
LIN {X 0,Y 420.367,Z 1204.581,A -85,B 0,C 180,E1 16478.266,E2 16478.266} C_VEL
LIN {X 0,Y 421.395,Z 1195.686,A -85,B 0,C 180,E1 16484.537,E2 16484.537} C_VEL
LIN {X 0,Y 424.341,Z 1180.719,A -85,B 0,C 180,E1 16491.26,E2 16491.26} C_VEL
LIN {X 0,Y 424.527,Z 1179.817,A -85,B 0,C 180,E1 16491.61,E2 16491.61} C_VEL
LIN {X 0,Y 422.13,Z 1174.079,A -85,B 0,C 180,E1 16493.833,E2 16493.833} C_VEL
LIN {X 0,Y 420.296,Z 1167.634,A -85,B 0,C 180,E1 16496.041,E2 16496.041} C_VEL
LIN {X 0,Y 428.485,Z 1143.19,A -85,B 0,C 180,E1 16502.534,E2 16502.534} C_VEL
LIN {X 0,Y 439.619,Z 1113.27,A -85,B 0,C 180,E1 16508.473,E2 16508.473} C_VEL
LIN {X 0,Y 452.513,Z 1079.993,A -85,B 0,C 180,E1 16513.53,E2 16513.53} C_VEL
LIN {X 0,Y 466.897,Z 1041.399,A -85,B 0,C 180,E1 16517.956,E2 16517.956} C_VEL
LIN {X 0,Y 481.074,Z 1000.346,A -85,B 0,C 180,E1 16521.522,E2 16521.522} C_VEL
LIN {X 0,Y 494.393,Z 955.627,A -85,B 0,C 180,E1 16524.367,E2 16524.367} C_VEL
LIN {X 0,Y 504.765,Z 913.482,A -85,B 0,C 180,E1 16526.337,E2 16526.337} C_VEL
LIN {X 0,Y 505.418,Z 909.825,A -85,B 0,C 180,E1 16526.515,E2 16526.515} C_VEL
LIN {X 0,Y 493.02,Z 879.681,A -85,B 0,C 180,E1 16530.94,E2 16530.94} C_VEL
LIN {X 0,Y 479.299,Z 853.071,A -85,B 0,C 180,E1 16535.908,E2 16535.908} C_VEL
LIN {X 0,Y 467.648,Z 834.013,A -85,B 0,C 180,E1 16540.658,E2 16540.658} C_VEL
LIN {X 0,Y 458.836,Z 820.979,A -85,B 0,C 180,E1 16545.081,E2 16545.081} C_VEL
LIN {X 0,Y 454.466,Z 814.631,A -85,B 0,C 180,E1 16547.797,E2 16547.797} C_VEL
LIN {X 0,Y 450.204,Z 808.102,A -85,B 0,C 180,E1 16551.302,E2 16551.302} C_VEL
LIN {X 0,Y 446.375,Z 801.821,A -85,B 0,C 180,E1 16556.957,E2 16556.957} C_VEL
LIN {X 0,Y 446.355,Z 801.485,A -85,B 0,C 180,E1 16563.385,E2 16563.385} C_VEL
LIN {X 0,Y 449.379,Z 807.644,A -85,B 0,C 180,E1 16568.447,E2 16568.447} C_VEL
LIN {X 0,Y 451.101,Z 809.806,A -85,B 0,C 180,E1 16570.085,E2 16570.085} C_VEL
LIN {X 0,Y 456.146,Z 817.53,A -85,B 0,C 180,E1 16573.864,E2 16573.864} C_VEL
LIN {X 0,Y 461.23,Z 825.387,A -85,B 0,C 180,E1 16576.948,E2 16576.948} C_VEL
LIN {X 0,Y 469.232,Z 837.77,A -85,B 0,C 180,E1 16580.85,E2 16580.85} C_VEL
LIN {X 0,Y 479.934,Z 856.543,A -85,B 0,C 180,E1 16585.389,E2 16585.389} C_VEL
LIN {X 0,Y 491.986,Z 882.223,A -85,B 0,C 180,E1 16590.18,E2 16590.18} C_VEL
LIN {X 0,Y 501.945,Z 910.037,A -85,B 0,C 180,E1 16594.345,E2 16594.345} C_VEL
LIN {X 0,Y 489.598,Z 957.802,A -85,B 0,C 180,E1 16597.054,E2 16597.054} C_VEL
LIN {X 0,Y 476.677,Z 997.844,A -85,B 0,C 180,E1 16600.039,E2 16600.039} C_VEL
LIN {X 0,Y 461.66,Z 1038.448,A -85,B 0,C 180,E1 16604.104,E2 16604.104} C_VEL
LIN {X 0,Y 448.316,Z 1072.317,A -85,B 0,C 180,E1 16608.588,E2 16608.588} C_VEL
LIN {X 0,Y 435.416,Z 1103.959,A -85,B 0,C 180,E1 16614.125,E2 16614.125} C_VEL
LIN {X 0,Y 425.413,Z 1130.021,A -85,B 0,C 180,E1 16620.18,E2 16620.18} C_VEL
LIN {X 0,Y 418.011,Z 1151.812,A -85,B 0,C 180,E1 16627.055,E2 16627.055} C_VEL
LIN {X 0,Y 414.517,Z 1165.507,A -85,B 0,C 180,E1 16633.045,E2 16633.045} C_VEL
LIN {X 0,Y 412.754,Z 1175.262,A -85,B 0,C 180,E1 16639.453,E2 16639.453} C_VEL
LIN {X 0,Y 412.201,Z 1180.418,A -85,B 0,C 180,E1 16645.796,E2 16645.796} C_VEL
LIN {X 0,Y 412.316,Z 1181.481,A -85,B 0,C 180,E1 16650.001,E2 16650.001} C_VEL
LIN {X 0,Y 412.341,Z 1179.155,A -85,B 0,C 180,E1 16656.313,E2 16656.313} C_VEL
LIN {X 0,Y 412.97,Z 1173.874,A -85,B 0,C 180,E1 16661.611,E2 16661.611} C_VEL
LIN {X 0,Y 415.059,Z 1163.12,A -85,B 0,C 180,E1 16668.014,E2 16668.014} C_VEL
LIN {X 0,Y 419.413,Z 1147.292,A -85,B 0,C 180,E1 16674.479,E2 16674.479} C_VEL
LIN {X 0,Y 426.921,Z 1125.631,A -85,B 0,C 180,E1 16680.881,E2 16680.881} C_VEL
LIN {X 0,Y 438.29,Z 1096.948,A -85,B 0,C 180,E1 16687.165,E2 16687.165} C_VEL
LIN {X 0,Y 451.471,Z 1064.25,A -85,B 0,C 180,E1 16692.487,E2 16692.487} C_VEL
LIN {X 0,Y 465.56,Z 1028.51,A -85,B 0,C 180,E1 16696.913,E2 16696.913} C_VEL
LIN {X 0,Y 479.563,Z 989.037,A -85,B 0,C 180,E1 16700.589,E2 16700.589} C_VEL
LIN {X 0,Y 493.389,Z 944.454,A -85,B 0,C 180,E1 16703.696,E2 16703.696} C_VEL
LIN {X 0,Y 502.055,Z 910.136,A -85,B 0,C 180,E1 16705.521,E2 16705.521} C_VEL
LIN {X 0,Y 491.161,Z 880.436,A -85,B 0,C 180,E1 16710.019,E2 16710.019} C_VEL
LIN {X 0,Y 479.209,Z 855.496,A -85,B 0,C 180,E1 16714.758,E2 16714.758} C_VEL
LIN {X 0,Y 467.693,Z 834.905,A -85,B 0,C 180,E1 16719.752,E2 16719.752} C_VEL
LIN {X 0,Y 458.259,Z 820.865,A -85,B 0,C 180,E1 16724.579,E2 16724.579} C_VEL
LIN {X 0,Y 453.992,Z 814.422,A -85,B 0,C 180,E1 16727.369,E2 16727.369} C_VEL
LIN {X 0,Y 449.822,Z 807.943,A -85,B 0,C 180,E1 16730.847,E2 16730.847} C_VEL
LIN {X 0,Y 446.266,Z 801.915,A -85,B 0,C 180,E1 16736.007,E2 16736.007} C_VEL
LIN {X 0,Y 446.23,Z 801.288,A -85,B 0,C 180,E1 16743.165,E2 16743.165} C_VEL
LIN {X 0,Y 449.459,Z 807.683,A -85,B 0,C 180,E1 16748.225,E2 16748.225} C_VEL
LIN {X 0,Y 451.259,Z 809.722,A -85,B 0,C 180,E1 16749.851,E2 16749.851} C_VEL
LIN {X 0,Y 456.518,Z 817.543,A -85,B 0,C 180,E1 16753.651,E2 16753.651} C_VEL
LIN {X 0,Y 462.467,Z 826.219,A -85,B 0,C 180,E1 16756.919,E2 16756.919} C_VEL
LIN {X 0,Y 472.517,Z 841.366,A -85,B 0,C 180,E1 16761.449,E2 16761.449} C_VEL
LIN {X 0,Y 485.494,Z 864.405,A -85,B 0,C 180,E1 16766.4,E2 16766.4} C_VEL
LIN {X 0,Y 498.068,Z 891.044,A -85,B 0,C 180,E1 16770.848,E2 16770.848} C_VEL
LIN {X 0,Y 505.346,Z 909.653,A -85,B 0,C 180,E1 16773.475,E2 16773.475} C_VEL
LIN {X 0,Y 493.251,Z 959.448,A -85,B 0,C 180,E1 16775.837,E2 16775.837} C_VEL
LIN {X 0,Y 480.477,Z 1002.027,A -85,B 0,C 180,E1 16778.617,E2 16778.617} C_VEL
LIN {X 0,Y 465.097,Z 1046.36,A -85,B 0,C 180,E1 16782.546,E2 16782.546} C_VEL
LIN {X 0,Y 451.853,Z 1081.721,A -85,B 0,C 180,E1 16786.718,E2 16786.718} C_VEL
LIN {X 0,Y 438.013,Z 1117.566,A -85,B 0,C 180,E1 16792.277,E2 16792.277} C_VEL
LIN {X 0,Y 427.335,Z 1146.159,A -85,B 0,C 180,E1 16798.173,E2 16798.173} C_VEL
LIN {X 0,Y 419.817,Z 1169.123,A -85,B 0,C 180,E1 16804.408,E2 16804.408} C_VEL
LIN {X 0,Y 415.095,Z 1187.403,A -85,B 0,C 180,E1 16811.19,E2 16811.19} C_VEL
LIN {X 0,Y 413.003,Z 1198.88,A -85,B 0,C 180,E1 16817.317,E2 16817.317} C_VEL
LIN {X 0,Y 412.304,Z 1206.094,A -85,B 0,C 180,E1 16823.686,E2 16823.686} C_VEL
LIN {X 0,Y 412.422,Z 1208.553,A -85,B 0,C 180,E1 16829.999,E2 16829.999} C_VEL
LIN {X 0,Y 412.332,Z 1206.098,A -85,B 0,C 180,E1 16836.311,E2 16836.311} C_VEL
LIN {X 0,Y 412.991,Z 1198.883,A -85,B 0,C 180,E1 16842.681,E2 16842.681} C_VEL
LIN {X 0,Y 415.212,Z 1186.732,A -85,B 0,C 180,E1 16849.119,E2 16849.119} C_VEL
LIN {X 0,Y 419.839,Z 1169.132,A -85,B 0,C 180,E1 16855.588,E2 16855.588} C_VEL
LIN {X 0,Y 420.296,Z 1167.634,A -85,B 0,C 180,E1 16856.041,E2 16856.041} C_VEL
LIN {X 0,Y 418.775,Z 1161.008,A -85,B 0,C 180,E1 16858.236,E2 16858.236} C_VEL
LIN {X 0,Y 417.394,Z 1153.85,A -85,B 0,C 180,E1 16860.438,E2 16860.438} C_VEL
LIN {X 0,Y 427.236,Z 1127.868,A -85,B 0,C 180,E1 16866.381,E2 16866.381} C_VEL
LIN {X 0,Y 440.379,Z 1094.993,A -85,B 0,C 180,E1 16872.094,E2 16872.094} C_VEL
LIN {X 0,Y 454.619,Z 1058.949,A -85,B 0,C 180,E1 16876.816,E2 16876.816} C_VEL
LIN {X 0,Y 469.784,Z 1018.448,A -85,B 0,C 180,E1 16880.812,E2 16880.812} C_VEL
LIN {X 0,Y 483.282,Z 977.573,A -85,B 0,C 180,E1 16883.823,E2 16883.823} C_VEL
LIN {X 0,Y 496.178,Z 930.506,A -85,B 0,C 180,E1 16886.397,E2 16886.397} C_VEL
LIN {X 0,Y 500.01,Z 913.18,A -85,B 0,C 180,E1 16887.166,E2 16887.166} C_VEL
LIN {X 0,Y 488.08,Z 883.424,A -85,B 0,C 180,E1 16891.714,E2 16891.714} C_VEL
LIN {X 0,Y 475.452,Z 858.413,A -85,B 0,C 180,E1 16896.561,E2 16896.561} C_VEL
LIN {X 0,Y 464.898,Z 840.614,A -85,B 0,C 180,E1 16901.146,E2 16901.146} C_VEL
LIN {X 0,Y 457.107,Z 828.52,A -85,B 0,C 180,E1 16905.268,E2 16905.268} C_VEL
LIN {X 0,Y 452.704,Z 821.964,A -85,B 0,C 180,E1 16908.185,E2 16908.185} C_VEL
LIN {X 0,Y 448.803,Z 815.801,A -85,B 0,C 180,E1 16911.519,E2 16911.519} C_VEL
LIN {X 0,Y 445.167,Z 809.411,A -85,B 0,C 180,E1 16917.192,E2 16917.192} C_VEL
LIN {X 0,Y 445.178,Z 809.572,A -85,B 0,C 180,E1 16923.394,E2 16923.394} C_VEL
LIN {X 0,Y 448.497,Z 815.658,A -85,B 0,C 180,E1 16928.708,E2 16928.708} C_VEL
LIN {X 0,Y 449.991,Z 818.249,A -85,B 0,C 180,E1 16930.193,E2 16930.193} C_VEL
LIN {X 0,Y 454.305,Z 825.136,A -85,B 0,C 180,E1 16933.686,E2 16933.686} C_VEL
LIN {X 0,Y 461.904,Z 836.483,A -85,B 0,C 180,E1 16938.124,E2 16938.124} C_VEL
LIN {X 0,Y 472.722,Z 855.647,A -85,B 0,C 180,E1 16943.35,E2 16943.35} C_VEL
LIN {X 0,Y 483.429,Z 877.668,A -85,B 0,C 180,E1 16947.946,E2 16947.946} C_VEL
LIN {X 0,Y 493.177,Z 902.822,A -85,B 0,C 180,E1 16952.15,E2 16952.15} C_VEL
LIN {X 0,Y 496.719,Z 914.145,A -85,B 0,C 180,E1 16953.811,E2 16953.811} C_VEL
LIN {X 0,Y 483.7,Z 961.744,A -85,B 0,C 180,E1 16956.531,E2 16956.531} C_VEL
LIN {X 0,Y 470.369,Z 1001.129,A -85,B 0,C 180,E1 16959.555,E2 16959.555} C_VEL
LIN {X 0,Y 455.158,Z 1040.975,A -85,B 0,C 180,E1 16963.631,E2 16963.631} C_VEL
LIN {X 0,Y 440.798,Z 1075.728,A -85,B 0,C 180,E1 16968.38,E2 16968.38} C_VEL
LIN {X 0,Y 427.83,Z 1106.604,A -85,B 0,C 180,E1 16973.961,E2 16973.961} C_VEL
LIN {X 0,Y 417.674,Z 1131.839,A -85,B 0,C 180,E1 16980.058,E2 16980.058} C_VEL
LIN {X 0,Y 410.183,Z 1153.203,A -85,B 0,C 180,E1 16987.024,E2 16987.024} C_VEL
LIN {X 0,Y 406.347,Z 1167.644,A -85,B 0,C 180,E1 16993.806,E2 16993.806} C_VEL
LIN {X 0,Y 404.75,Z 1176.691,A -85,B 0,C 180,E1 17000.329,E2 17000.329} C_VEL
LIN {X 0,Y 404.32,Z 1180.677,A -85,B 0,C 180,E1 17005.714,E2 17005.714} C_VEL
LIN {X 0,Y 404.44,Z 1181.74,A -85,B 0,C 180,E1 17010.001,E2 17010.001} C_VEL
LIN {X 0,Y 404.45,Z 1179.417,A -85,B 0,C 180,E1 17016.437,E2 17016.437} C_VEL
LIN {X 0,Y 405.13,Z 1174.138,A -85,B 0,C 180,E1 17021.839,E2 17021.839} C_VEL
LIN {X 0,Y 407.306,Z 1163.559,A -85,B 0,C 180,E1 17028.283,E2 17028.283} C_VEL
LIN {X 0,Y 411.961,Z 1147.563,A -85,B 0,C 180,E1 17034.951,E2 17034.951} C_VEL
LIN {X 0,Y 419.853,Z 1125.904,A -85,B 0,C 180,E1 17041.459,E2 17041.459} C_VEL
LIN {X 0,Y 431.053,Z 1098.794,A -85,B 0,C 180,E1 17047.513,E2 17047.513} C_VEL
LIN {X 0,Y 444.406,Z 1066.991,A -85,B 0,C 180,E1 17052.85,E2 17052.85} C_VEL
LIN {X 0,Y 459.602,Z 1029.827,A -85,B 0,C 180,E1 17057.538,E2 17057.538} C_VEL
LIN {X 0,Y 474.114,Z 990.377,A -85,B 0,C 180,E1 17061.255,E2 17061.255} C_VEL
LIN {X 0,Y 488.473,Z 945.492,A -85,B 0,C 180,E1 17064.411,E2 17064.411} C_VEL
LIN {X 0,Y 496.692,Z 915.053,A -85,B 0,C 180,E1 17066.002,E2 17066.002} C_VEL
LIN {X 0,Y 488.294,Z 889.347,A -85,B 0,C 180,E1 17069.897,E2 17069.897} C_VEL
LIN {X 0,Y 476.702,Z 863.6,A -85,B 0,C 180,E1 17074.741,E2 17074.741} C_VEL
LIN {X 0,Y 466.687,Z 845.267,A -85,B 0,C 180,E1 17079.211,E2 17079.211} C_VEL
LIN {X 0,Y 458.994,Z 832.604,A -85,B 0,C 180,E1 17083.211,E2 17083.211} C_VEL
LIN {X 0,Y 452.458,Z 822.154,A -85,B 0,C 180,E1 17087.464,E2 17087.464} C_VEL
LIN {X 0,Y 448.529,Z 815.676,A -85,B 0,C 180,E1 17090.971,E2 17090.971} C_VEL
LIN {X 0,Y 445.043,Z 809.506,A -85,B 0,C 180,E1 17096.24,E2 17096.24} C_VEL
LIN {X 0,Y 445.08,Z 809.478,A -85,B 0,C 180,E1 17103.234,E2 17103.234} C_VEL
LIN {X 0,Y 448.593,Z 815.654,A -85,B 0,C 180,E1 17108.485,E2 17108.485} C_VEL
LIN {X 0,Y 450.186,Z 818.281,A -85,B 0,C 180,E1 17109.989,E2 17109.989} C_VEL
LIN {X 0,Y 455.025,Z 825.35,A -85,B 0,C 180,E1 17113.513,E2 17113.513} C_VEL
LIN {X 0,Y 462.609,Z 836.518,A -85,B 0,C 180,E1 17117.78,E2 17117.78} C_VEL
LIN {X 0,Y 474.089,Z 855.933,A -85,B 0,C 180,E1 17122.927,E2 17122.927} C_VEL
LIN {X 0,Y 486.615,Z 880.223,A -85,B 0,C 180,E1 17127.77,E2 17127.77} C_VEL
LIN {X 0,Y 498.614,Z 909.315,A -85,B 0,C 180,E1 17132.293,E2 17132.293} C_VEL
LIN {X 0,Y 499.887,Z 914.552,A -85,B 0,C 180,E1 17132.94,E2 17132.94} C_VEL
LIN {X 0,Y 488.003,Z 961.222,A -85,B 0,C 180,E1 17135.181,E2 17135.181} C_VEL
LIN {X 0,Y 474.614,Z 1004.04,A -85,B 0,C 180,E1 17138.025,E2 17138.025} C_VEL
LIN {X 0,Y 459.219,Z 1047.018,A -85,B 0,C 180,E1 17141.882,E2 17141.882} C_VEL
LIN {X 0,Y 445.091,Z 1083.25,A -85,B 0,C 180,E1 17146.236,E2 17146.236} C_VEL
LIN {X 0,Y 431.009,Z 1118.425,A -85,B 0,C 180,E1 17151.799,E2 17151.799} C_VEL
LIN {X 0,Y 419.658,Z 1147.517,A -85,B 0,C 180,E1 17157.971,E2 17157.971} C_VEL
LIN {X 0,Y 411.858,Z 1170.604,A -85,B 0,C 180,E1 17164.461,E2 17164.461} C_VEL
LIN {X 0,Y 407.282,Z 1187.47,A -85,B 0,C 180,E1 17170.976,E2 17170.976} C_VEL
LIN {X 0,Y 405.156,Z 1198.616,A -85,B 0,C 180,E1 17177.068,E2 17177.068} C_VEL
LIN {X 0,Y 404.409,Z 1205.833,A -85,B 0,C 180,E1 17183.563,E2 17183.563} C_VEL
LIN {X 0,Y 404.525,Z 1208.294,A -85,B 0,C 180,E1 17189.999,E2 17189.999} C_VEL
LIN {X 0,Y 404.435,Z 1205.837,A -85,B 0,C 180,E1 17196.435,E2 17196.435} C_VEL
LIN {X 0,Y 405.143,Z 1198.619,A -85,B 0,C 180,E1 17202.931,E2 17202.931} C_VEL
LIN {X 0,Y 407.504,Z 1186.465,A -85,B 0,C 180,E1 17209.495,E2 17209.495} C_VEL
LIN {X 0,Y 412.587,Z 1168.328,A -85,B 0,C 180,E1 17216.247,E2 17216.247} C_VEL
LIN {X 0,Y 417.394,Z 1153.85,A -85,B 0,C 180,E1 17220.438,E2 17220.438} C_VEL
LIN {X 0,Y 416.44,Z 1146.423,A -85,B 0,C 180,E1 17222.625,E2 17222.625} C_VEL
LIN {X 0,Y 416.107,Z 1138.317,A -85,B 0,C 180,E1 17224.766,E2 17224.766} C_VEL
LIN {X 0,Y 429.014,Z 1107.298,A -85,B 0,C 180,E1 17230.818,E2 17230.818} C_VEL
LIN {X 0,Y 442.939,Z 1073.7,A -85,B 0,C 180,E1 17235.759,E2 17235.759} C_VEL
LIN {X 0,Y 458.482,Z 1034.696,A -85,B 0,C 180,E1 17240.103,E2 17240.103} C_VEL
LIN {X 0,Y 473.391,Z 992.857,A -85,B 0,C 180,E1 17243.571,E2 17243.571} C_VEL
LIN {X 0,Y 487.754,Z 945.865,A -85,B 0,C 180,E1 17246.426,E2 17246.426} C_VEL
LIN {X 0,Y 494.919,Z 917.441,A -85,B 0,C 180,E1 17247.712,E2 17247.712} C_VEL
LIN {X 0,Y 484.245,Z 889.564,A -85,B 0,C 180,E1 17252.082,E2 17252.082} C_VEL
LIN {X 0,Y 472.119,Z 864.641,A -85,B 0,C 180,E1 17257.032,E2 17257.032} C_VEL
LIN {X 0,Y 462.293,Z 847.367,A -85,B 0,C 180,E1 17261.556,E2 17261.556} C_VEL
LIN {X 0,Y 454.773,Z 835.523,A -85,B 0,C 180,E1 17265.713,E2 17265.713} C_VEL
LIN {X 0,Y 450.96,Z 829.524,A -85,B 0,C 180,E1 17268.392,E2 17268.392} C_VEL
LIN {X 0,Y 447.453,Z 823.502,A -85,B 0,C 180,E1 17271.677,E2 17271.677} C_VEL
LIN {X 0,Y 443.974,Z 817.091,A -85,B 0,C 180,E1 17277.368,E2 17277.368} C_VEL
LIN {X 0,Y 444.023,Z 817.59,A -85,B 0,C 180,E1 17283.433,E2 17283.433} C_VEL
LIN {X 0,Y 447.153,Z 823.436,A -85,B 0,C 180,E1 17288.735,E2 17288.735} C_VEL
LIN {X 0,Y 452.469,Z 832.725,A -85,B 0,C 180,E1 17293.507,E2 17293.507} C_VEL
LIN {X 0,Y 459.449,Z 843.814,A -85,B 0,C 180,E1 17297.884,E2 17297.884} C_VEL
LIN {X 0,Y 469.391,Z 862.044,A -85,B 0,C 180,E1 17302.961,E2 17302.961} C_VEL
LIN {X 0,Y 480.192,Z 885.377,A -85,B 0,C 180,E1 17307.875,E2 17307.875} C_VEL
LIN {X 0,Y 489.593,Z 911.438,A -85,B 0,C 180,E1 17312.236,E2 17312.236} C_VEL
LIN {X 0,Y 491.421,Z 918.427,A -85,B 0,C 180,E1 17313.261,E2 17313.261} C_VEL
LIN {X 0,Y 478.593,Z 963.217,A -85,B 0,C 180,E1 17315.837,E2 17315.837} C_VEL
LIN {X 0,Y 464.319,Z 1003.901,A -85,B 0,C 180,E1 17319.017,E2 17319.017} C_VEL
LIN {X 0,Y 449.176,Z 1042.233,A -85,B 0,C 180,E1 17322.995,E2 17322.995} C_VEL
LIN {X 0,Y 434.712,Z 1075.993,A -85,B 0,C 180,E1 17327.664,E2 17327.664} C_VEL
LIN {X 0,Y 420.754,Z 1107.984,A -85,B 0,C 180,E1 17333.531,E2 17333.531} C_VEL
LIN {X 0,Y 409.924,Z 1133.655,A -85,B 0,C 180,E1 17339.93,E2 17339.93} C_VEL
LIN {X 0,Y 402.645,Z 1153.471,A -85,B 0,C 180,E1 17346.568,E2 17346.568} C_VEL
LIN {X 0,Y 398.597,Z 1167.908,A -85,B 0,C 180,E1 17353.482,E2 17353.482} C_VEL
LIN {X 0,Y 396.889,Z 1176.952,A -85,B 0,C 180,E1 17360.136,E2 17360.136} C_VEL
LIN {X 0,Y 396.419,Z 1180.937,A -85,B 0,C 180,E1 17365.629,E2 17365.629} C_VEL
LIN {X 0,Y 396.541,Z 1181.999,A -85,B 0,C 180,E1 17370.001,E2 17370.001} C_VEL
LIN {X 0,Y 396.56,Z 1179.678,A -85,B 0,C 180,E1 17376.565,E2 17376.565} C_VEL
LIN {X 0,Y 397.286,Z 1174.402,A -85,B 0,C 180,E1 17382.076,E2 17382.076} C_VEL
LIN {X 0,Y 399.495,Z 1164.279,A -85,B 0,C 180,E1 17388.421,E2 17388.421} C_VEL
LIN {X 0,Y 404.554,Z 1147.833,A -85,B 0,C 180,E1 17395.44,E2 17395.44} C_VEL
LIN {X 0,Y 412.82,Z 1126.295,A -85,B 0,C 180,E1 17402.024,E2 17402.024} C_VEL
LIN {X 0,Y 424.776,Z 1098.612,A -85,B 0,C 180,E1 17408.279,E2 17408.279} C_VEL
LIN {X 0,Y 438.484,Z 1067.261,A -85,B 0,C 180,E1 17413.572,E2 17413.572} C_VEL
LIN {X 0,Y 454.142,Z 1030.065,A -85,B 0,C 180,E1 17418.302,E2 17418.302} C_VEL
LIN {X 0,Y 469.223,Z 990.359,A -85,B 0,C 180,E1 17422.045,E2 17422.045} C_VEL
LIN {X 0,Y 483.915,Z 945.589,A -85,B 0,C 180,E1 17425.19,E2 17425.19} C_VEL
LIN {X 0,Y 491.492,Z 917.923,A -85,B 0,C 180,E1 17426.665,E2 17426.665} C_VEL
LIN {X 0,Y 481.838,Z 889.457,A -85,B 0,C 180,E1 17431.277,E2 17431.277} C_VEL
LIN {X 0,Y 470.647,Z 864.786,A -85,B 0,C 180,E1 17436.29,E2 17436.29} C_VEL
LIN {X 0,Y 461.401,Z 847.732,A -85,B 0,C 180,E1 17440.835,E2 17440.835} C_VEL
LIN {X 0,Y 453.988,Z 835.295,A -85,B 0,C 180,E1 17445.249,E2 17445.249} C_VEL
LIN {X 0,Y 450.319,Z 829.333,A -85,B 0,C 180,E1 17447.901,E2 17447.901} C_VEL
LIN {X 0,Y 446.827,Z 823.202,A -85,B 0,C 180,E1 17451.291,E2 17451.291} C_VEL
LIN {X 0,Y 443.828,Z 817.097,A -85,B 0,C 180,E1 17456.474,E2 17456.474} C_VEL
LIN {X 0,Y 443.889,Z 817.452,A -85,B 0,C 180,E1 17463.182,E2 17463.182} C_VEL
LIN {X 0,Y 447.704,Z 823.657,A -85,B 0,C 180,E1 17468.746,E2 17468.746} C_VEL
LIN {X 0,Y 453.415,Z 833.347,A -85,B 0,C 180,E1 17473.501,E2 17473.501} C_VEL
LIN {X 0,Y 460.771,Z 844.494,A -85,B 0,C 180,E1 17477.695,E2 17477.695} C_VEL
LIN {X 0,Y 471.376,Z 863.178,A -85,B 0,C 180,E1 17482.695,E2 17482.695} C_VEL
LIN {X 0,Y 482.817,Z 886.233,A -85,B 0,C 180,E1 17487.364,E2 17487.364} C_VEL
LIN {X 0,Y 494.135,Z 915.281,A -85,B 0,C 180,E1 17491.987,E2 17491.987} C_VEL
LIN {X 0,Y 494.487,Z 918.865,A -85,B 0,C 180,E1 17492.347,E2 17492.347} C_VEL
LIN {X 0,Y 482.317,Z 964.753,A -85,B 0,C 180,E1 17494.614,E2 17494.614} C_VEL
LIN {X 0,Y 467.23,Z 1010.492,A -85,B 0,C 180,E1 17497.769,E2 17497.769} C_VEL
LIN {X 0,Y 451.994,Z 1051.173,A -85,B 0,C 180,E1 17501.579,E2 17501.579} C_VEL
LIN {X 0,Y 436.354,Z 1089.594,A -85,B 0,C 180,E1 17506.418,E2 17506.418} C_VEL
LIN {X 0,Y 422.839,Z 1121.991,A -85,B 0,C 180,E1 17511.844,E2 17511.844} C_VEL
LIN {X 0,Y 411.359,Z 1150.58,A -85,B 0,C 180,E1 17518.184,E2 17518.184} C_VEL
LIN {X 0,Y 403.747,Z 1172.3,A -85,B 0,C 180,E1 17524.655,E2 17524.655} C_VEL
LIN {X 0,Y 399.031,Z 1189.609,A -85,B 0,C 180,E1 17531.738,E2 17531.738} C_VEL
LIN {X 0,Y 397.099,Z 1199.96,A -85,B 0,C 180,E1 17537.918,E2 17537.918} C_VEL
LIN {X 0,Y 396.506,Z 1205.572,A -85,B 0,C 180,E1 17543.434,E2 17543.434} C_VEL
LIN {X 0,Y 396.627,Z 1208.035,A -85,B 0,C 180,E1 17549.999,E2 17549.999} C_VEL
LIN {X 0,Y 396.53,Z 1205.576,A -85,B 0,C 180,E1 17556.564,E2 17556.564} C_VEL
LIN {X 0,Y 397.31,Z 1198.355,A -85,B 0,C 180,E1 17563.19,E2 17563.19} C_VEL
LIN {X 0,Y 399.828,Z 1186.198,A -85,B 0,C 180,E1 17569.885,E2 17569.885} C_VEL
LIN {X 0,Y 405.033,Z 1168.593,A -85,B 0,C 180,E1 17576.595,E2 17576.595} C_VEL
LIN {X 0,Y 414.032,Z 1143.75,A -85,B 0,C 180,E1 17583.505,E2 17583.505} C_VEL
LIN {X 0,Y 416.107,Z 1138.317,A -85,B 0,C 180,E1 17584.766,E2 17584.766} C_VEL
LIN {X 0,Y 416.242,Z 1130.044,A -85,B 0,C 180,E1 17586.878,E2 17586.878} C_VEL
LIN {X 0,Y 416.622,Z 1121.166,A -85,B 0,C 180,E1 17588.975,E2 17588.975} C_VEL
LIN {X 0,Y 430.346,Z 1089.394,A -85,B 0,C 180,E1 17594.343,E2 17594.343} C_VEL
LIN {X 0,Y 446.599,Z 1050.984,A -85,B 0,C 180,E1 17599.206,E2 17599.206} C_VEL
LIN {X 0,Y 461.957,Z 1011.355,A -85,B 0,C 180,E1 17602.943,E2 17602.943} C_VEL
LIN {X 0,Y 477.381,Z 966.067,A -85,B 0,C 180,E1 17606.083,E2 17606.083} C_VEL
LIN {X 0,Y 489.253,Z 923.201,A -85,B 0,C 180,E1 17608.255,E2 17608.255} C_VEL
LIN {X 0,Y 489.696,Z 921.104,A -85,B 0,C 180,E1 17608.352,E2 17608.352} C_VEL
LIN {X 0,Y 479.612,Z 894.024,A -85,B 0,C 180,E1 17612.73,E2 17612.73} C_VEL
LIN {X 0,Y 467.969,Z 869.429,A -85,B 0,C 180,E1 17617.819,E2 17617.819} C_VEL
LIN {X 0,Y 457.542,Z 850.405,A -85,B 0,C 180,E1 17623.073,E2 17623.073} C_VEL
LIN {X 0,Y 449.654,Z 837.527,A -85,B 0,C 180,E1 17628.231,E2 17628.231} C_VEL
LIN {X 0,Y 445.594,Z 831.068,A -85,B 0,C 180,E1 17632.01,E2 17632.01} C_VEL
LIN {X 0,Y 442.518,Z 824.487,A -85,B 0,C 180,E1 17638.032,E2 17638.032} C_VEL
LIN {X 0,Y 442.589,Z 825.368,A -85,B 0,C 180,E1 17643.322,E2 17643.322} C_VEL
LIN {X 0,Y 445.674,Z 831.212,A -85,B 0,C 180,E1 17648.764,E2 17648.764} C_VEL
LIN {X 0,Y 450.64,Z 840.564,A -85,B 0,C 180,E1 17653.439,E2 17653.439} C_VEL
LIN {X 0,Y 457.138,Z 851.463,A -85,B 0,C 180,E1 17657.728,E2 17657.728} C_VEL
LIN {X 0,Y 466.413,Z 869.206,A -85,B 0,C 180,E1 17662.738,E2 17662.738} C_VEL
LIN {X 0,Y 476.743,Z 892.638,A -85,B 0,C 180,E1 17667.722,E2 17667.722} C_VEL
LIN {X 0,Y 485.809,Z 920.369,A -85,B 0,C 180,E1 17672.399,E2 17672.399} C_VEL
LIN {X 0,Y 485.614,Z 924.198,A -85,B 0,C 180,E1 17672.742,E2 17672.742} C_VEL
LIN {X 0,Y 472.162,Z 968.447,A -85,B 0,C 180,E1 17675.389,E2 17675.389} C_VEL
LIN {X 0,Y 456.852,Z 1010.413,A -85,B 0,C 180,E1 17678.803,E2 17678.803} C_VEL
LIN {X 0,Y 441.58,Z 1047.246,A -85,B 0,C 180,E1 17682.813,E2 17682.813} C_VEL
LIN {X 0,Y 425.949,Z 1082.304,A -85,B 0,C 180,E1 17687.911,E2 17687.911} C_VEL
LIN {X 0,Y 413.084,Z 1110.553,A -85,B 0,C 180,E1 17693.372,E2 17693.372} C_VEL
LIN {X 0,Y 401.622,Z 1136.822,A -85,B 0,C 180,E1 17700.193,E2 17700.193} C_VEL
LIN {X 0,Y 394.669,Z 1155.191,A -85,B 0,C 180,E1 17706.719,E2 17706.719} C_VEL
LIN {X 0,Y 390.85,Z 1168.173,A -85,B 0,C 180,E1 17713.145,E2 17713.145} C_VEL
LIN {X 0,Y 389.03,Z 1177.213,A -85,B 0,C 180,E1 17719.934,E2 17719.934} C_VEL
LIN {X 0,Y 388.541,Z 1181.196,A -85,B 0,C 180,E1 17725.54,E2 17725.54} C_VEL
LIN {X 0,Y 388.643,Z 1182.258,A -85,B 0,C 180,E1 17730.001,E2 17730.001} C_VEL
LIN {X 0,Y 388.699,Z 1179.938,A -85,B 0,C 180,E1 17736.699,E2 17736.699} C_VEL
LIN {X 0,Y 389.461,Z 1174.665,A -85,B 0,C 180,E1 17742.323,E2 17742.323} C_VEL
LIN {X 0,Y 392.236,Z 1163.107,A -85,B 0,C 180,E1 17749.53,E2 17749.53} C_VEL
LIN {X 0,Y 397.798,Z 1146.605,A -85,B 0,C 180,E1 17756.511,E2 17756.511} C_VEL
LIN {X 0,Y 407.435,Z 1123.154,A -85,B 0,C 180,E1 17763.517,E2 17763.517} C_VEL
LIN {X 0,Y 419.372,Z 1096.787,A -85,B 0,C 180,E1 17769.392,E2 17769.392} C_VEL
LIN {X 0,Y 434.141,Z 1064.087,A -85,B 0,C 180,E1 17774.818,E2 17774.818} C_VEL
LIN {X 0,Y 449.807,Z 1027.889,A -85,B 0,C 180,E1 17779.338,E2 17779.338} C_VEL
LIN {X 0,Y 465.265,Z 987.981,A -85,B 0,C 180,E1 17783.046,E2 17783.046} C_VEL
LIN {X 0,Y 479.425,Z 945.697,A -85,B 0,C 180,E1 17785.987,E2 17785.987} C_VEL
LIN {X 0,Y 486.082,Z 921.292,A -85,B 0,C 180,E1 17787.347,E2 17787.347} C_VEL
LIN {X 0,Y 477.159,Z 894.077,A -85,B 0,C 180,E1 17791.912,E2 17791.912} C_VEL
LIN {X 0,Y 466.723,Z 870.196,A -85,B 0,C 180,E1 17796.939,E2 17796.939} C_VEL
LIN {X 0,Y 458.229,Z 853.836,A -85,B 0,C 180,E1 17801.446,E2 17801.446} C_VEL
LIN {X 0,Y 451.612,Z 842.403,A -85,B 0,C 180,E1 17805.603,E2 17805.603} C_VEL
LIN {X 0,Y 448.06,Z 836.312,A -85,B 0,C 180,E1 17808.462,E2 17808.462} C_VEL
LIN {X 0,Y 445.147,Z 830.852,A -85,B 0,C 180,E1 17811.461,E2 17811.461} C_VEL
LIN {X 0,Y 442.306,Z 824.491,A -85,B 0,C 180,E1 17817.074,E2 17817.074} C_VEL
LIN {X 0,Y 442.546,Z 825.31,A -85,B 0,C 180,E1 17823.131,E2 17823.131} C_VEL
LIN {X 0,Y 446.715,Z 832.943,A -85,B 0,C 180,E1 17829.379,E2 17829.379} C_VEL
LIN {X 0,Y 451.545,Z 840.934,A -85,B 0,C 180,E1 17833.311,E2 17833.311} C_VEL
LIN {X 0,Y 458.349,Z 851.791,A -85,B 0,C 180,E1 17837.455,E2 17837.455} C_VEL
LIN {X 0,Y 468.504,Z 870.353,A -85,B 0,C 180,E1 17842.467,E2 17842.467} C_VEL
LIN {X 0,Y 479.437,Z 893.633,A -85,B 0,C 180,E1 17847.227,E2 17847.227} C_VEL
LIN {X 0,Y 489.614,Z 921.119,A -85,B 0,C 180,E1 17851.654,E2 17851.654} C_VEL
LIN {X 0,Y 477.226,Z 966.133,A -85,B 0,C 180,E1 17853.915,E2 17853.915} C_VEL
LIN {X 0,Y 461.831,Z 1011.435,A -85,B 0,C 180,E1 17857.065,E2 17857.065} C_VEL
LIN {X 0,Y 446.555,Z 1050.891,A -85,B 0,C 180,E1 17860.785,E2 17860.785} C_VEL
LIN {X 0,Y 430.377,Z 1089.317,A -85,B 0,C 180,E1 17865.655,E2 17865.655} C_VEL
LIN {X 0,Y 416.304,Z 1121.715,A -85,B 0,C 180,E1 17871.134,E2 17871.134} C_VEL
LIN {X 0,Y 404.194,Z 1150.596,A -85,B 0,C 180,E1 17877.635,E2 17877.635} C_VEL
LIN {X 0,Y 396.217,Z 1172.224,A -85,B 0,C 180,E1 17884.214,E2 17884.214} C_VEL
LIN {X 0,Y 391.307,Z 1189.341,A -85,B 0,C 180,E1 17891.364,E2 17891.364} C_VEL
LIN {X 0,Y 389.242,Z 1199.696,A -85,B 0,C 180,E1 17897.67,E2 17897.67} C_VEL
LIN {X 0,Y 388.62,Z 1205.311,A -85,B 0,C 180,E1 17903.3,E2 17903.3} C_VEL
LIN {X 0,Y 388.729,Z 1207.775,A -85,B 0,C 180,E1 17909.999,E2 17909.999} C_VEL
LIN {X 0,Y 388.641,Z 1205.315,A -85,B 0,C 180,E1 17916.697,E2 17916.697} C_VEL
LIN {X 0,Y 389.479,Z 1198.092,A -85,B 0,C 180,E1 17923.46,E2 17923.46} C_VEL
LIN {X 0,Y 392.137,Z 1185.93,A -85,B 0,C 180,E1 17930.292,E2 17930.292} C_VEL
LIN {X 0,Y 397.622,Z 1168.322,A -85,B 0,C 180,E1 17937.131,E2 17937.131} C_VEL
LIN {X 0,Y 407.408,Z 1142.622,A -85,B 0,C 180,E1 17944.372,E2 17944.372} C_VEL
LIN {X 0,Y 416.622,Z 1121.166,A -85,B 0,C 180,E1 17948.975,E2 17948.975} C_VEL
LIN {X 0,Y 417.392,Z 1112.107,A -85,B 0,C 180,E1 17951.037,E2 17951.037} C_VEL
LIN {X 0,Y 418.42,Z 1102.451,A -85,B 0,C 180,E1 17953.041,E2 17953.041} C_VEL
LIN {X 0,Y 434.958,Z 1065.379,A -85,B 0,C 180,E1 17958.328,E2 17958.328} C_VEL
LIN {X 0,Y 450.886,Z 1027.269,A -85,B 0,C 180,E1 17962.35,E2 17962.35} C_VEL
LIN {X 0,Y 466.236,Z 985.809,A -85,B 0,C 180,E1 17965.638,E2 17965.638} C_VEL
LIN {X 0,Y 479.959,Z 941.717,A -85,B 0,C 180,E1 17968.218,E2 17968.218} C_VEL
LIN {X 0,Y 484.291,Z 924.179,A -85,B 0,C 180,E1 17969.104,E2 17969.104} C_VEL
LIN {X 0,Y 474.717,Z 897.808,A -85,B 0,C 180,E1 17973.527,E2 17973.527} C_VEL
LIN {X 0,Y 463.623,Z 873.643,A -85,B 0,C 180,E1 17978.731,E2 17978.731} C_VEL
LIN {X 0,Y 454.343,Z 856.625,A -85,B 0,C 180,E1 17983.747,E2 17983.747} C_VEL
LIN {X 0,Y 447.617,Z 844.897,A -85,B 0,C 180,E1 17988.55,E2 17988.55} C_VEL
LIN {X 0,Y 443.936,Z 838.693,A -85,B 0,C 180,E1 17992.164,E2 17992.164} C_VEL
LIN {X 0,Y 441.025,Z 832.249,A -85,B 0,C 180,E1 17998.025,E2 17998.025} C_VEL
LIN {X 0,Y 441.065,Z 833.237,A -85,B 0,C 180,E1 18003.303,E2 18003.303} C_VEL
LIN {X 0,Y 444.535,Z 840.47,A -85,B 0,C 180,E1 18009.403,E2 18009.403} C_VEL
LIN {X 0,Y 448.688,Z 848.475,A -85,B 0,C 180,E1 18013.436,E2 18013.436} C_VEL
LIN {X 0,Y 454.892,Z 859.39,A -85,B 0,C 180,E1 18017.694,E2 18017.694} C_VEL
LIN {X 0,Y 463.224,Z 875.988,A -85,B 0,C 180,E1 18022.437,E2 18022.437} C_VEL
LIN {X 0,Y 472.562,Z 898.505,A -85,B 0,C 180,E1 18027.334,E2 18027.334} C_VEL
LIN {X 0,Y 480.609,Z 924.135,A -85,B 0,C 180,E1 18031.765,E2 18031.765} C_VEL
LIN {X 0,Y 480.505,Z 927.669,A -85,B 0,C 180,E1 18032.105,E2 18032.105} C_VEL
LIN {X 0,Y 465.996,Z 973.099,A -85,B 0,C 180,E1 18034.899,E2 18034.899} C_VEL
LIN {X 0,Y 450.516,Z 1013.981,A -85,B 0,C 180,E1 18038.308,E2 18038.308} C_VEL
LIN {X 0,Y 433.86,Z 1052.354,A -85,B 0,C 180,E1 18042.653,E2 18042.653} C_VEL
LIN {X 0,Y 418.288,Z 1086.004,A -85,B 0,C 180,E1 18047.741,E2 18047.741} C_VEL
LIN {X 0,Y 403.948,Z 1116.092,A -85,B 0,C 180,E1 18053.902,E2 18053.902} C_VEL
LIN {X 0,Y 393.838,Z 1138.687,A -85,B 0,C 180,E1 18060.081,E2 18060.081} C_VEL
LIN {X 0,Y 386.588,Z 1157.136,A -85,B 0,C 180,E1 18066.992,E2 18066.992} C_VEL
LIN {X 0,Y 382.681,Z 1170.3,A -85,B 0,C 180,E1 18073.955,E2 18073.955} C_VEL
LIN {X 0,Y 381.049,Z 1178.613,A -85,B 0,C 180,E1 18080.874,E2 18080.874} C_VEL
LIN {X 0,Y 380.582,Z 1182.206,A -85,B 0,C 180,E1 18087.726,E2 18087.726} C_VEL
LIN {X 0,Y 380.716,Z 1182.188,A -85,B 0,C 180,E1 18092.276,E2 18092.276} C_VEL
LIN {X 0,Y 381.139,Z 1178.534,A -85,B 0,C 180,E1 18099.126,E2 18099.126} C_VEL
LIN {X 0,Y 382.704,Z 1170.148,A -85,B 0,C 180,E1 18106.046,E2 18106.046} C_VEL
LIN {X 0,Y 386.729,Z 1156.922,A -85,B 0,C 180,E1 18113.002,E2 18113.002} C_VEL
LIN {X 0,Y 393.965,Z 1138.41,A -85,B 0,C 180,E1 18119.911,E2 18119.911} C_VEL
LIN {X 0,Y 405.232,Z 1113.382,A -85,B 0,C 180,E1 18126.631,E2 18126.631} C_VEL
LIN {X 0,Y 419.218,Z 1083.989,A -85,B 0,C 180,E1 18132.506,E2 18132.506} C_VEL
LIN {X 0,Y 435.508,Z 1048.605,A -85,B 0,C 180,E1 18137.738,E2 18137.738} C_VEL
LIN {X 0,Y 451.386,Z 1011.45,A -85,B 0,C 180,E1 18141.839,E2 18141.839} C_VEL
LIN {X 0,Y 467.881,Z 967.763,A -85,B 0,C 180,E1 18145.372,E2 18145.372} C_VEL
LIN {X 0,Y 480.932,Z 925.313,A -85,B 0,C 180,E1 18147.939,E2 18147.939} C_VEL
LIN {X 0,Y 472.593,Z 898.971,A -85,B 0,C 180,E1 18152.486,E2 18152.486} C_VEL
LIN {X 0,Y 462.675,Z 875.064,A -85,B 0,C 180,E1 18157.696,E2 18157.696} C_VEL
LIN {X 0,Y 453.566,Z 856.901,A -85,B 0,C 180,E1 18163.003,E2 18163.003} C_VEL
LIN {X 0,Y 446.504,Z 844.417,A -85,B 0,C 180,E1 18168.235,E2 18168.235} C_VEL
LIN {X 0,Y 443.421,Z 838.461,A -85,B 0,C 180,E1 18171.684,E2 18171.684} C_VEL
LIN {X 0,Y 440.815,Z 832.252,A -85,B 0,C 180,E1 18177.064,E2 18177.064} C_VEL
LIN {X 0,Y 441.004,Z 833.036,A -85,B 0,C 180,E1 18183.019,E2 18183.019} C_VEL
LIN {X 0,Y 445.021,Z 840.606,A -85,B 0,C 180,E1 18189.23,E2 18189.23} C_VEL
LIN {X 0,Y 449.515,Z 848.448,A -85,B 0,C 180,E1 18193.136,E2 18193.136} C_VEL
LIN {X 0,Y 456.122,Z 859.623,A -85,B 0,C 180,E1 18197.357,E2 18197.357} C_VEL
LIN {X 0,Y 465.266,Z 876.991,A -85,B 0,C 180,E1 18202.129,E2 18202.129} C_VEL
LIN {X 0,Y 475.745,Z 900.349,A -85,B 0,C 180,E1 18206.97,E2 18206.97} C_VEL
LIN {X 0,Y 484.34,Z 925.496,A -85,B 0,C 180,E1 18211.042,E2 18211.042} C_VEL
LIN {X 0,Y 471.447,Z 969.832,A -85,B 0,C 180,E1 18213.342,E2 18213.342} C_VEL
LIN {X 0,Y 455.836,Z 1014.222,A -85,B 0,C 180,E1 18216.493,E2 18216.493} C_VEL
LIN {X 0,Y 439.361,Z 1054.905,A -85,B 0,C 180,E1 18220.457,E2 18220.457} C_VEL
LIN {X 0,Y 423.141,Z 1092.083,A -85,B 0,C 180,E1 18225.311,E2 18225.311} C_VEL
LIN {X 0,Y 407.798,Z 1125.882,A -85,B 0,C 180,E1 18231.294,E2 18231.294} C_VEL
LIN {X 0,Y 396.072,Z 1152.967,A -85,B 0,C 180,E1 18237.714,E2 18237.714} C_VEL
LIN {X 0,Y 387.889,Z 1174.498,A -85,B 0,C 180,E1 18244.624,E2 18244.624} C_VEL
LIN {X 0,Y 383.264,Z 1190.364,A -85,B 0,C 180,E1 18251.613,E2 18251.613} C_VEL
LIN {X 0,Y 381.193,Z 1200.79,A -85,B 0,C 180,E1 18258.567,E2 18258.567} C_VEL
LIN {X 0,Y 380.727,Z 1205.05,A -85,B 0,C 180,E1 18263.16,E2 18263.16} C_VEL
LIN {X 0,Y 380.831,Z 1207.516,A -85,B 0,C 180,E1 18269.999,E2 18269.999} C_VEL
LIN {X 0,Y 380.754,Z 1205.055,A -85,B 0,C 180,E1 18276.837,E2 18276.837} C_VEL
LIN {X 0,Y 381.671,Z 1197.828,A -85,B 0,C 180,E1 18283.741,E2 18283.741} C_VEL
LIN {X 0,Y 384.473,Z 1185.662,A -85,B 0,C 180,E1 18290.714,E2 18290.714} C_VEL
LIN {X 0,Y 390.215,Z 1168.049,A -85,B 0,C 180,E1 18297.69,E2 18297.69} C_VEL
LIN {X 0,Y 400.482,Z 1142.509,A -85,B 0,C 180,E1 18305.005,E2 18305.005} C_VEL
LIN {X 0,Y 413.44,Z 1113.367,A -85,B 0,C 180,E1 18311.138,E2 18311.138} C_VEL
LIN {X 0,Y 418.42,Z 1102.451,A -85,B 0,C 180,E1 18313.041,E2 18313.041} C_VEL
LIN {X 0,Y 419.859,Z 1092.597,A -85,B 0,C 180,E1 18315.002,E2 18315.002} C_VEL
LIN {X 0,Y 421.753,Z 1082.081,A -85,B 0,C 180,E1 18316.91,E2 18316.91} C_VEL
LIN {X 0,Y 438.127,Z 1045.586,A -85,B 0,C 180,E1 18321.368,E2 18321.368} C_VEL
LIN {X 0,Y 455.812,Z 1001.509,A -85,B 0,C 180,E1 18325.343,E2 18325.343} C_VEL
LIN {X 0,Y 470.91,Z 957.776,A -85,B 0,C 180,E1 18328.176,E2 18328.176} C_VEL
LIN {X 0,Y 479.231,Z 928.381,A -85,B 0,C 180,E1 18329.693,E2 18329.693} C_VEL
LIN {X 0,Y 470.02,Z 902.105,A -85,B 0,C 180,E1 18334.267,E2 18334.267} C_VEL
LIN {X 0,Y 459.861,Z 879.273,A -85,B 0,C 180,E1 18339.368,E2 18339.368} C_VEL
LIN {X 0,Y 451.68,Z 863.45,A -85,B 0,C 180,E1 18344.155,E2 18344.155} C_VEL
LIN {X 0,Y 445.172,Z 852.045,A -85,B 0,C 180,E1 18348.982,E2 18348.982} C_VEL
LIN {X 0,Y 442.034,Z 846.268,A -85,B 0,C 180,E1 18352.402,E2 18352.402} C_VEL
LIN {X 0,Y 439.531,Z 840.016,A -85,B 0,C 180,E1 18358.019,E2 18358.019} C_VEL
LIN {X 0,Y 439.491,Z 840.942,A -85,B 0,C 180,E1 18363.191,E2 18363.191} C_VEL
LIN {X 0,Y 442.521,Z 848.058,A -85,B 0,C 180,E1 18369.26,E2 18369.26} C_VEL
LIN {X 0,Y 446.741,Z 856.367,A -85,B 0,C 180,E1 18373.434,E2 18373.434} C_VEL
LIN {X 0,Y 452.368,Z 867.063,A -85,B 0,C 180,E1 18377.608,E2 18377.608} C_VEL
LIN {X 0,Y 460.107,Z 883.339,A -85,B 0,C 180,E1 18382.3,E2 18382.3} C_VEL
LIN {X 0,Y 469.057,Z 906.34,A -85,B 0,C 180,E1 18387.312,E2 18387.312} C_VEL
LIN {X 0,Y 475.721,Z 928.993,A -85,B 0,C 180,E1 18391.287,E2 18391.287} C_VEL
LIN {X 0,Y 460.77,Z 975.201,A -85,B 0,C 180,E1 18394.21,E2 18394.21} C_VEL
LIN {X 0,Y 445.379,Z 1014.619,A -85,B 0,C 180,E1 18397.527,E2 18397.527} C_VEL
LIN {X 0,Y 428.412,Z 1052.496,A -85,B 0,C 180,E1 18401.831,E2 18401.831} C_VEL
LIN {X 0,Y 412.151,Z 1086.498,A -85,B 0,C 180,E1 18407.018,E2 18407.018} C_VEL
LIN {X 0,Y 397.097,Z 1116.862,A -85,B 0,C 180,E1 18413.323,E2 18413.323} C_VEL
LIN {X 0,Y 385.926,Z 1140.651,A -85,B 0,C 180,E1 18420.052,E2 18420.052} C_VEL
LIN {X 0,Y 378.153,Z 1160,A -85,B 0,C 180,E1 18427.691,E2 18427.691} C_VEL
LIN {X 0,Y 374.49,Z 1172.236,A -85,B 0,C 180,E1 18434.749,E2 18434.749} C_VEL
LIN {X 0,Y 373.17,Z 1178.875,A -85,B 0,C 180,E1 18440.68,E2 18440.68} C_VEL
LIN {X 0,Y 372.7,Z 1182.465,A -85,B 0,C 180,E1 18447.677,E2 18447.677} C_VEL
LIN {X 0,Y 372.825,Z 1182.447,A -85,B 0,C 180,E1 18452.324,E2 18452.324} C_VEL
LIN {X 0,Y 373.253,Z 1178.797,A -85,B 0,C 180,E1 18459.321,E2 18459.321} C_VEL
LIN {X 0,Y 374.957,Z 1170.414,A -85,B 0,C 180,E1 18466.387,E2 18466.387} C_VEL
LIN {X 0,Y 379.765,Z 1155.841,A -85,B 0,C 180,E1 18474.097,E2 18474.097} C_VEL
LIN {X 0,Y 388.024,Z 1136.121,A -85,B 0,C 180,E1 18481.292,E2 18481.292} C_VEL
LIN {X 0,Y 400.452,Z 1110.126,A -85,B 0,C 180,E1 18488.165,E2 18488.165} C_VEL
LIN {X 0,Y 415.264,Z 1079.832,A -85,B 0,C 180,E1 18494.022,E2 18494.022} C_VEL
LIN {X 0,Y 432.247,Z 1044.365,A -85,B 0,C 180,E1 18499.114,E2 18499.114} C_VEL
LIN {X 0,Y 449.447,Z 1004.465,A -85,B 0,C 180,E1 18503.311,E2 18503.311} C_VEL
LIN {X 0,Y 465.207,Z 962.777,A -85,B 0,C 180,E1 18506.553,E2 18506.553} C_VEL
LIN {X 0,Y 475.728,Z 929.012,A -85,B 0,C 180,E1 18508.596,E2 18508.596} C_VEL
LIN {X 0,Y 467.966,Z 903.484,A -85,B 0,C 180,E1 18513.139,E2 18513.139} C_VEL
LIN {X 0,Y 458.873,Z 880.661,A -85,B 0,C 180,E1 18518.259,E2 18518.259} C_VEL
LIN {X 0,Y 450.436,Z 863.475,A -85,B 0,C 180,E1 18523.508,E2 18523.508} C_VEL
LIN {X 0,Y 444.455,Z 851.966,A -85,B 0,C 180,E1 18528.367,E2 18528.367} C_VEL
LIN {X 0,Y 441.467,Z 846.054,A -85,B 0,C 180,E1 18531.809,E2 18531.809} C_VEL
LIN {X 0,Y 439.314,Z 840.025,A -85,B 0,C 180,E1 18537.054,E2 18537.054} C_VEL
LIN {X 0,Y 439.463,Z 840.768,A -85,B 0,C 180,E1 18542.906,E2 18542.906} C_VEL
LIN {X 0,Y 443.1,Z 848.22,A -85,B 0,C 180,E1 18549.085,E2 18549.085} C_VEL
LIN {X 0,Y 447.519,Z 856.255,A -85,B 0,C 180,E1 18553.099,E2 18553.099} C_VEL
LIN {X 0,Y 454.092,Z 867.914,A -85,B 0,C 180,E1 18557.437,E2 18557.437} C_VEL
LIN {X 0,Y 462.908,Z 885.315,A -85,B 0,C 180,E1 18562.2,E2 18562.2} C_VEL
LIN {X 0,Y 473.381,Z 910.781,A -85,B 0,C 180,E1 18567.397,E2 18567.397} C_VEL
LIN {X 0,Y 479.104,Z 929.439,A -85,B 0,C 180,E1 18570.413,E2 18570.413} C_VEL
LIN {X 0,Y 465.387,Z 974.541,A -85,B 0,C 180,E1 18572.82,E2 18572.82} C_VEL
LIN {X 0,Y 449.815,Z 1017.027,A -85,B 0,C 180,E1 18575.917,E2 18575.917} C_VEL
LIN {X 0,Y 432.284,Z 1058.624,A -85,B 0,C 180,E1 18580.081,E2 18580.081} C_VEL
LIN {X 0,Y 416.691,Z 1093.029,A -85,B 0,C 180,E1 18584.702,E2 18584.702} C_VEL
LIN {X 0,Y 401.275,Z 1125.795,A -85,B 0,C 180,E1 18590.592,E2 18590.592} C_VEL
LIN {X 0,Y 389.064,Z 1152.692,A -85,B 0,C 180,E1 18597.059,E2 18597.059} C_VEL
LIN {X 0,Y 380.458,Z 1174.227,A -85,B 0,C 180,E1 18604.093,E2 18604.093} C_VEL
LIN {X 0,Y 375.545,Z 1190.096,A -85,B 0,C 180,E1 18611.221,E2 18611.221} C_VEL
LIN {X 0,Y 373.325,Z 1200.526,A -85,B 0,C 180,E1 18618.322,E2 18618.322} C_VEL
LIN {X 0,Y 372.842,Z 1204.789,A -85,B 0,C 180,E1 18623.015,E2 18623.015} C_VEL
LIN {X 0,Y 372.933,Z 1207.257,A -85,B 0,C 180,E1 18629.999,E2 18629.999} C_VEL
LIN {X 0,Y 372.862,Z 1204.794,A -85,B 0,C 180,E1 18636.982,E2 18636.982} C_VEL
LIN {X 0,Y 373.867,Z 1197.565,A -85,B 0,C 180,E1 18644.034,E2 18644.034} C_VEL
LIN {X 0,Y 376.82,Z 1185.394,A -85,B 0,C 180,E1 18651.155,E2 18651.155} C_VEL
LIN {X 0,Y 382.881,Z 1167.778,A -85,B 0,C 180,E1 18658.267,E2 18658.267} C_VEL
LIN {X 0,Y 393.46,Z 1142.679,A -85,B 0,C 180,E1 18665.589,E2 18665.589} C_VEL
LIN {X 0,Y 406.506,Z 1114.575,A -85,B 0,C 180,E1 18671.64,E2 18671.64} C_VEL
LIN {X 0,Y 421.753,Z 1082.081,A -85,B 0,C 180,E1 18676.91,E2 18676.91} C_VEL
LIN {X 0,Y 423.884,Z 1071.421,A -85,B 0,C 180,E1 18678.781,E2 18678.781} C_VEL
LIN {X 0,Y 425.619,Z 1061.744,A -85,B 0,C 180,E1 18680.373,E2 18680.373} C_VEL
LIN {X 0,Y 426.268,Z 1060.18,A -85,B 0,C 180,E1 18680.56,E2 18680.56} C_VEL
LIN {X 0,Y 444.724,Z 1017.815,A -85,B 0,C 180,E1 18684.845,E2 18684.845} C_VEL
LIN {X 0,Y 460.442,Z 976.367,A -85,B 0,C 180,E1 18687.899,E2 18687.899} C_VEL
LIN {X 0,Y 474.137,Z 932.519,A -85,B 0,C 180,E1 18690.29,E2 18690.29} C_VEL
LIN {X 0,Y 465.394,Z 906.328,A -85,B 0,C 180,E1 18695.024,E2 18695.024} C_VEL
LIN {X 0,Y 455.814,Z 884.039,A -85,B 0,C 180,E1 18700.221,E2 18700.221} C_VEL
LIN {X 0,Y 447.022,Z 866.343,A -85,B 0,C 180,E1 18705.929,E2 18705.929} C_VEL
LIN {X 0,Y 442.244,Z 858.357,A -85,B 0,C 180,E1 18709.904,E2 18709.904} C_VEL
LIN {X 0,Y 440.007,Z 853.807,A -85,B 0,C 180,E1 18712.59,E2 18712.59} C_VEL
LIN {X 0,Y 437.749,Z 847.704,A -85,B 0,C 180,E1 18718.011,E2 18718.011} C_VEL
LIN {X 0,Y 437.612,Z 848.512,A -85,B 0,C 180,E1 18723.019,E2 18723.019} C_VEL
LIN {X 0,Y 440.55,Z 855.775,A -85,B 0,C 180,E1 18729.177,E2 18729.177} C_VEL
LIN {X 0,Y 444.565,Z 864.266,A -85,B 0,C 180,E1 18733.501,E2 18733.501} C_VEL
LIN {X 0,Y 451.375,Z 877.583,A -85,B 0,C 180,E1 18738.53,E2 18738.53} C_VEL
LIN {X 0,Y 459.562,Z 897.151,A -85,B 0,C 180,E1 18743.726,E2 18743.726} C_VEL
LIN {X 0,Y 467.502,Z 921.204,A -85,B 0,C 180,E1 18748.634,E2 18748.634} C_VEL
LIN {X 0,Y 470.292,Z 934.305,A -85,B 0,C 180,E1 18750.79,E2 18750.79} C_VEL
LIN {X 0,Y 454.385,Z 980.735,A -85,B 0,C 180,E1 18753.758,E2 18753.758} C_VEL
LIN {X 0,Y 438.102,Z 1020.179,A -85,B 0,C 180,E1 18757.233,E2 18757.233} C_VEL
LIN {X 0,Y 420.798,Z 1057.409,A -85,B 0,C 180,E1 18761.622,E2 18761.622} C_VEL
LIN {X 0,Y 404.047,Z 1090.774,A -85,B 0,C 180,E1 18766.973,E2 18766.973} C_VEL
LIN {X 0,Y 389.273,Z 1119.725,A -85,B 0,C 180,E1 18773.231,E2 18773.231} C_VEL
LIN {X 0,Y 378.033,Z 1142.611,A -85,B 0,C 180,E1 18780.024,E2 18780.024} C_VEL
LIN {X 0,Y 370.188,Z 1161.569,A -85,B 0,C 180,E1 18787.832,E2 18787.832} C_VEL
LIN {X 0,Y 366.7,Z 1172.559,A -85,B 0,C 180,E1 18794.465,E2 18794.465} C_VEL
LIN {X 0,Y 365.304,Z 1179.136,A -85,B 0,C 180,E1 18800.477,E2 18800.477} C_VEL
LIN {X 0,Y 364.8,Z 1182.724,A -85,B 0,C 180,E1 18807.627,E2 18807.627} C_VEL
LIN {X 0,Y 364.922,Z 1182.707,A -85,B 0,C 180,E1 18812.374,E2 18812.374} C_VEL
LIN {X 0,Y 365.373,Z 1179.059,A -85,B 0,C 180,E1 18819.524,E2 18819.524} C_VEL
LIN {X 0,Y 367.232,Z 1170.679,A -85,B 0,C 180,E1 18826.742,E2 18826.742} C_VEL
LIN {X 0,Y 372.302,Z 1156.163,A -85,B 0,C 180,E1 18834.585,E2 18834.585} C_VEL
LIN {X 0,Y 380.527,Z 1137.464,A -85,B 0,C 180,E1 18841.604,E2 18841.604} C_VEL
LIN {X 0,Y 393.401,Z 1111.573,A -85,B 0,C 180,E1 18848.624,E2 18848.624} C_VEL
LIN {X 0,Y 408.108,Z 1082.798,A -85,B 0,C 180,E1 18854.361,E2 18854.361} C_VEL
LIN {X 0,Y 425.085,Z 1048.447,A -85,B 0,C 180,E1 18859.452,E2 18859.452} C_VEL
LIN {X 0,Y 441.602,Z 1011.887,A -85,B 0,C 180,E1 18863.502,E2 18863.502} C_VEL
LIN {X 0,Y 459.126,Z 967.765,A -85,B 0,C 180,E1 18867.063,E2 18867.063} C_VEL
LIN {X 0,Y 470.502,Z 932.831,A -85,B 0,C 180,E1 18869.229,E2 18869.229} C_VEL
LIN {X 0,Y 463.228,Z 907.669,A -85,B 0,C 180,E1 18873.887,E2 18873.887} C_VEL
LIN {X 0,Y 454.71,Z 885.698,A -85,B 0,C 180,E1 18879.037,E2 18879.037} C_VEL
LIN {X 0,Y 447.372,Z 869.939,A -85,B 0,C 180,E1 18884.022,E2 18884.022} C_VEL
LIN {X 0,Y 441.892,Z 858.859,A -85,B 0,C 180,E1 18888.923,E2 18888.923} C_VEL
LIN {X 0,Y 439.36,Z 853.514,A -85,B 0,C 180,E1 18892.105,E2 18892.105} C_VEL
LIN {X 0,Y 437.254,Z 847.567,A -85,B 0,C 180,E1 18898.031,E2 18898.031} C_VEL
LIN {X 0,Y 437.611,Z 848.484,A -85,B 0,C 180,E1 18902.825,E2 18902.825} C_VEL
LIN {X 0,Y 441.068,Z 855.815,A -85,B 0,C 180,E1 18908.941,E2 18908.941} C_VEL
LIN {X 0,Y 445.743,Z 864.416,A -85,B 0,C 180,E1 18913.238,E2 18913.238} C_VEL
LIN {X 0,Y 452.954,Z 878.027,A -85,B 0,C 180,E1 18918.172,E2 18918.172} C_VEL
LIN {X 0,Y 461.758,Z 897.322,A -85,B 0,C 180,E1 18923.131,E2 18923.131} C_VEL
LIN {X 0,Y 470.534,Z 920.878,A -85,B 0,C 180,E1 18927.762,E2 18927.762} C_VEL
LIN {X 0,Y 474.03,Z 932.837,A -85,B 0,C 180,E1 18929.747,E2 18929.747} C_VEL
LIN {X 0,Y 460.409,Z 976.158,A -85,B 0,C 180,E1 18932.091,E2 18932.091} C_VEL
LIN {X 0,Y 444.666,Z 1017.66,A -85,B 0,C 180,E1 18935.141,E2 18935.141} C_VEL
LIN {X 0,Y 425.91,Z 1060.837,A -85,B 0,C 180,E1 18939.521,E2 18939.521} C_VEL
LIN {X 0,Y 409.328,Z 1095.906,A -85,B 0,C 180,E1 18944.39,E2 18944.39} C_VEL
LIN {X 0,Y 393.392,Z 1128.584,A -85,B 0,C 180,E1 18950.458,E2 18950.458} C_VEL
LIN {X 0,Y 381.174,Z 1154.407,A -85,B 0,C 180,E1 18956.967,E2 18956.967} C_VEL
LIN {X 0,Y 372.481,Z 1175.524,A -85,B 0,C 180,E1 18964.142,E2 18964.142} C_VEL
LIN {X 0,Y 367.795,Z 1190.031,A -85,B 0,C 180,E1 18970.925,E2 18970.925} C_VEL
LIN {X 0,Y 365.479,Z 1200.263,A -85,B 0,C 180,E1 18978.068,E2 18978.068} C_VEL
LIN {X 0,Y 364.869,Z 1205.151,A -85,B 0,C 180,E1 18983.761,E2 18983.761} C_VEL
LIN {X 0,Y 365.035,Z 1206.998,A -85,B 0,C 180,E1 18989.999,E2 18989.999} C_VEL
LIN {X 0,Y 364.958,Z 1204.533,A -85,B 0,C 180,E1 18997.134,E2 18997.134} C_VEL
LIN {X 0,Y 365.716,Z 1199.058,A -85,B 0,C 180,E1 19003.024,E2 19003.024} C_VEL
LIN {X 0,Y 368.467,Z 1187.485,A -85,B 0,C 180,E1 19010.4,E2 19010.4} C_VEL
LIN {X 0,Y 374.626,Z 1170.058,A -85,B 0,C 180,E1 19017.958,E2 19017.958} C_VEL
LIN {X 0,Y 384.289,Z 1147.745,A -85,B 0,C 180,E1 19024.9,E2 19024.9} C_VEL
LIN {X 0,Y 398.261,Z 1118.642,A -85,B 0,C 180,E1 19031.604,E2 19031.604} C_VEL
LIN {X 0,Y 414.255,Z 1085.655,A -85,B 0,C 180,E1 19037.191,E2 19037.191} C_VEL
LIN {X 0,Y 426.268,Z 1060.18,A -85,B 0,C 180,E1 19040.56,E2 19040.56} C_VEL
LIN {X 0,Y 428.991,Z 1048.698,A -85,B 0,C 180,E1 19042.274,E2 19042.274} C_VEL
LIN {X 0,Y 431.846,Z 1036.608,A -85,B 0,C 180,E1 19043.942,E2 19043.942} C_VEL
LIN {X 0,Y 448.517,Z 996.646,A -85,B 0,C 180,E1 19047.38,E2 19047.38} C_VEL
LIN {X 0,Y 464.965,Z 949.718,A -85,B 0,C 180,E1 19050.29,E2 19050.29} C_VEL
LIN {X 0,Y 468.807,Z 935.584,A -85,B 0,C 180,E1 19051.078,E2 19051.078} C_VEL
LIN {X 0,Y 460.897,Z 911.234,A -85,B 0,C 180,E1 19055.646,E2 19055.646} C_VEL
LIN {X 0,Y 452.6,Z 890.967,A -85,B 0,C 180,E1 19060.487,E2 19060.487} C_VEL
LIN {X 0,Y 444.406,Z 873.587,A -85,B 0,C 180,E1 19066.158,E2 19066.158} C_VEL
LIN {X 0,Y 439.907,Z 865.577,A -85,B 0,C 180,E1 19070.225,E2 19070.225} C_VEL
LIN {X 0,Y 437.961,Z 861.342,A -85,B 0,C 180,E1 19072.804,E2 19072.804} C_VEL
LIN {X 0,Y 435.674,Z 855.299,A -85,B 0,C 180,E1 19078.995,E2 19078.995} C_VEL
LIN {X 0,Y 435.736,Z 856.258,A -85,B 0,C 180,E1 19082.97,E2 19082.97} C_VEL
LIN {X 0,Y 438.281,Z 863.177,A -85,B 0,C 180,E1 19088.975,E2 19088.975} C_VEL
LIN {X 0,Y 443.425,Z 873.832,A -85,B 0,C 180,E1 19094.416,E2 19094.416} C_VEL
LIN {X 0,Y 450.761,Z 890.507,A -85,B 0,C 180,E1 19100.032,E2 19100.032} C_VEL
LIN {X 0,Y 458.796,Z 912.281,A -85,B 0,C 180,E1 19105.336,E2 19105.336} C_VEL
LIN {X 0,Y 465.373,Z 936.94,A -85,B 0,C 180,E1 19110.052,E2 19110.052} C_VEL
LIN {X 0,Y 449.967,Z 980.993,A -85,B 0,C 180,E1 19112.907,E2 19112.907} C_VEL
LIN {X 0,Y 433.439,Z 1019.977,A -85,B 0,C 180,E1 19116.327,E2 19116.327} C_VEL
LIN {X 0,Y 415.254,Z 1058.026,A -85,B 0,C 180,E1 19120.828,E2 19120.828} C_VEL
LIN {X 0,Y 398.232,Z 1090.745,A -85,B 0,C 180,E1 19126.109,E2 19126.109} C_VEL
LIN {X 0,Y 383.159,Z 1119.094,A -85,B 0,C 180,E1 19132.272,E2 19132.272} C_VEL
LIN {X 0,Y 371.624,Z 1141.587,A -85,B 0,C 180,E1 19138.935,E2 19138.935} C_VEL
LIN {X 0,Y 363.312,Z 1160.102,A -85,B 0,C 180,E1 19146.512,E2 19146.512} C_VEL
LIN {X 0,Y 359.475,Z 1171.092,A -85,B 0,C 180,E1 19152.888,E2 19152.888} C_VEL
LIN {X 0,Y 357.431,Z 1179.398,A -85,B 0,C 180,E1 19160.265,E2 19160.265} C_VEL
LIN {X 0,Y 356.899,Z 1182.984,A -85,B 0,C 180,E1 19167.575,E2 19167.575} C_VEL
LIN {X 0,Y 357.018,Z 1182.967,A -85,B 0,C 180,E1 19172.427,E2 19172.427} C_VEL
LIN {X 0,Y 357.497,Z 1179.322,A -85,B 0,C 180,E1 19179.735,E2 19179.735} C_VEL
LIN {X 0,Y 359.516,Z 1170.945,A -85,B 0,C 180,E1 19187.112,E2 19187.112} C_VEL
LIN {X 0,Y 364.876,Z 1156.433,A -85,B 0,C 180,E1 19195.12,E2 19195.12} C_VEL
LIN {X 0,Y 373.713,Z 1137.324,A -85,B 0,C 180,E1 19202.397,E2 19202.397} C_VEL
LIN {X 0,Y 387.595,Z 1110.672,A -85,B 0,C 180,E1 19209.675,E2 19209.675} C_VEL
LIN {X 0,Y 402.992,Z 1081.593,A -85,B 0,C 180,E1 19215.436,E2 19215.436} C_VEL
LIN {X 0,Y 420.661,Z 1047.093,A -85,B 0,C 180,E1 19220.509,E2 19220.509} C_VEL
LIN {X 0,Y 438.113,Z 1009.258,A -85,B 0,C 180,E1 19224.616,E2 19224.616} C_VEL
LIN {X 0,Y 455.641,Z 965.902,A -85,B 0,C 180,E1 19228.06,E2 19228.06} C_VEL
LIN {X 0,Y 465.353,Z 936.897,A -85,B 0,C 180,E1 19229.84,E2 19229.84} C_VEL
LIN {X 0,Y 458.561,Z 911.859,A -85,B 0,C 180,E1 19234.65,E2 19234.65} C_VEL
LIN {X 0,Y 450.582,Z 890.385,A -85,B 0,C 180,E1 19239.892,E2 19239.892} C_VEL
LIN {X 0,Y 443.097,Z 873.285,A -85,B 0,C 180,E1 19245.641,E2 19245.641} C_VEL
LIN {X 0,Y 437.81,Z 861.552,A -85,B 0,C 180,E1 19251.578,E2 19251.578} C_VEL
LIN {X 0,Y 435.416,Z 855.237,A -85,B 0,C 180,E1 19258.023,E2 19258.023} C_VEL
LIN {X 0,Y 435.735,Z 856.147,A -85,B 0,C 180,E1 19262.744,E2 19262.744} C_VEL
LIN {X 0,Y 439.009,Z 863.408,A -85,B 0,C 180,E1 19268.796,E2 19268.796} C_VEL
LIN {X 0,Y 443.378,Z 872.048,A -85,B 0,C 180,E1 19273.185,E2 19273.185} C_VEL
LIN {X 0,Y 449.639,Z 884.113,A -85,B 0,C 180,E1 19277.615,E2 19277.615} C_VEL
LIN {X 0,Y 458.121,Z 903.677,A -85,B 0,C 180,E1 19282.763,E2 19282.763} C_VEL
LIN {X 0,Y 466.376,Z 927.293,A -85,B 0,C 180,E1 19287.489,E2 19287.489} C_VEL
LIN {X 0,Y 468.752,Z 937.174,A -85,B 0,C 180,E1 19289.11,E2 19289.11} C_VEL
LIN {X 0,Y 454.403,Z 980.99,A -85,B 0,C 180,E1 19291.551,E2 19291.551} C_VEL
LIN {X 0,Y 437.331,Z 1023.663,A -85,B 0,C 180,E1 19294.833,E2 19294.833} C_VEL
LIN {X 0,Y 419.414,Z 1063.302,A -85,B 0,C 180,E1 19298.977,E2 19298.977} C_VEL
LIN {X 0,Y 401.18,Z 1100.255,A -85,B 0,C 180,E1 19304.301,E2 19304.301} C_VEL
LIN {X 0,Y 385.793,Z 1130.618,A -85,B 0,C 180,E1 19310.189,E2 19310.189} C_VEL
LIN {X 0,Y 372.373,Z 1158.111,A -85,B 0,C 180,E1 19317.472,E2 19317.472} C_VEL
LIN {X 0,Y 363.9,Z 1178.174,A -85,B 0,C 180,E1 19324.808,E2 19324.808} C_VEL
LIN {X 0,Y 359.465,Z 1191.804,A -85,B 0,C 180,E1 19331.772,E2 19331.772} C_VEL
LIN {X 0,Y 357.452,Z 1201.251,A -85,B 0,C 180,E1 19339.032,E2 19339.032} C_VEL
LIN {X 0,Y 356.98,Z 1205.562,A -85,B 0,C 180,E1 19345.142,E2 19345.142} C_VEL
LIN {X 0,Y 357.152,Z 1206.739,A -85,B 0,C 180,E1 19349.999,E2 19349.999} C_VEL
LIN {X 0,Y 357.055,Z 1204.272,A -85,B 0,C 180,E1 19357.293,E2 19357.293} C_VEL
LIN {X 0,Y 357.982,Z 1198.117,A -85,B 0,C 180,E1 19363.833,E2 19363.833} C_VEL
LIN {X 0,Y 361.187,Z 1186.037,A -85,B 0,C 180,E1 19371.473,E2 19371.473} C_VEL
LIN {X 0,Y 367.846,Z 1168.455,A -85,B 0,C 180,E1 19379.07,E2 19379.07} C_VEL
LIN {X 0,Y 379.347,Z 1143.494,A -85,B 0,C 180,E1 19386.691,E2 19386.691} C_VEL
LIN {X 0,Y 393.797,Z 1114.897,A -85,B 0,C 180,E1 19393.086,E2 19393.086} C_VEL
LIN {X 0,Y 411.532,Z 1079.766,A -85,B 0,C 180,E1 19398.853,E2 19398.853} C_VEL
